(* CODESYS project full_demo.190528.1.project

Project tree, tasks and I/O mapping:
  MIC7001 : Changsha Xiangji-ARM Cortex A9(xilinx zynq7000)-linux, Changsha Xiangji Hiden Technology Co.Ltd, version 3.5.10.40
    application Application
      libraries: Standard, * (System); CAA File, * (CAA Technical Workgroup); CAA Types Extern, * (CAA Technical Workgroup); CAA Callback Extern, * (CAA Technical Workgroup); SysMem, * (System); Util, 3.5.11.0 (System); SysFile, 3.5.9.0 (System); SysTypes Interfaces, * (System); CAN API, 1.0.0.3 (3S - Smart Software Solutions GmbH); SysTime, * (System); CAA DTUtil Extern, 3.5.12.0 (CAA Technical Workgroup); CAA SerialCom, 3.5.12.0 (CAA Technical Workgroup); cyber gpio, 3.5.10.40 (cyber); AC_DataLog, 3.5.13.0 (3S - Smart Software Solutions GmbH)
      task MainTask (cyclic, interval 20 ms, priority 15) calls prg_input, prg_engine, prg_pump, prg_output, prg_data
      task can_0 (cyclic, interval 8 ms, priority 10) calls prg_can0
      task VISU_TASK (cyclic, interval 100 ms, priority 31) calls VisuElems.Visu_Prg, prg_set_inmode, prg_heartbeat
      task EtherCAT_Task (cyclic, interval t#4ms, priority 1) calls nothing
      program prg_pump [ST]
      program prg_output [ST]
      program prg_input [ST]
      j1939/
        function temp_absZero_to_1735oC [ST]
        function block PGN_F004_RPM [ST]
        function pros100 [ST]
        function block PGN_FEEE_TEMP [ST]
        function temp_neg40_to_210oC [ST]
        function PACK [ST]
      program prg_can0 [CFC]: act_set_rpm, act_send_to_MID
      function_blocks/
        function block MsgProcessor_j1939_f004 [ST]: ProcessMessage
        function block fb_pp_avg [ST]
        function block MsgProcessor_j1939_f003 [ST]: ProcessMessage
        function block MsgProcessor_MID [ST]: ProcessMessage
        function block MsgProcessor_j1939_fef2 [ST]: ProcessMessage
        function block MsgProcessor_j1939_feef [ST]: ProcessMessage
        function block MsgProcessor_j1939_feee [ST]: ProcessMessage
      program prg_set_inmode [ST]
      ENUM/
        data type ENGINE_STATE
        data type STATE1939
        data type WORK_MODE
      global variables GVL
      parameters/
        function block FB_PARA_DINT [ST]: clear_all, rd_all, chk_chg, wr_all
        data type DUT_PARA_DINT
        data type DUT_PARA_REAL
        function block FB_PARA_REAL [ST]: rd_all, chk_chg, clear_all, wr_all
      functions/
        function fn_write_in_mode_file [ST]
        function fn_write_real_data [ST]
        function fn_read_in_mode_file [ST]
        function fn_get_Q_221ma [ST]
        function fn_get_Q_408ma [ST]
        function fn_get_Q_631ma [ST]
        function fn_get_Q_521ma [ST]
        function fn_write_dint_data [ST]
        function fn_get_mins [ST]
      program prg_data [ST]
      visualisation Visualization
      program prg_engine [ST]: get_x_rpm_set
      GPRS/
        function block File_Read [ST]
        function Iccid_Get [ST]
        program prg_heartbeat [ST]
        function block fb_get_iccid [ST]
        function block fb_m26 [ST]
        function block fb_get_lac [ST]
        function fn_cyber_layer1 [ST]
        function fn_cyber_layer2 [ST]
        function fn_cyber_heartBeat [ST]
        function fn_sn_str_to_byte [ST]
      gprs_lib/
        function block Com_Read [ST]
        function block reset_gprs [ST]
        function block Udp_Config [ST]
        function block Udp_Init [ST]
        function block UDP_Read [ST]
        function block Udp_Write [ST]
    EtherCAT_Master_SoftMotion : EtherCAT Master SoftMotion, 3S - Smart Software Solutions GmbH, version 3.5.13.30
        settings: NetworkName = 'eth0'; NetworkName = "eth0"; SelectNetworkByName = True
      MIR3502 : MIR3502, Cyber-MI, order no. MIR3502, version Revision=16#00000000
          settings: DC sync0 cycletime = 4000; DC sync1 cycletime = 4000
          unmapped channels: PWM00-C24, PWM01-C35, DO00-C01, DO01-C02, DO02-C03, DO03-C04, DO04-C05, DO05-C06, DO06-C07, DO07-C08, DO08-C09, DO09-C10, DO10-C11, DO11-C12, DO12-C35, DO13-C34, DO14-C33, DO15-C32, DO16-C31, DO17-C30, DO18-C29, DO19-C28, DO20-C27, DO21-C26, DO22-C25, DO23-C24, AI00-C20, AI01-C19, AI02-C18, AI03-C17, AI04-C16, AI05-C15, AI06-C01, AI07-C02, AI08-C03, AI09-C04, AI10-C05, AI11-C06, AI12-C07, AI13-C08,
            AI14-C09, AI15-C10, AI16-C11, AI17-C12, AI18-C35, AI19-C34, AI20-C33, AI21-C32, AI22-C31, AI23-C30, AI24-C29, AI25-C28, AI26-C27, AI27-C26, AI28-C25, AI29-C24, AI30-iPWM0, AI31-iPWM1, DI00-C20, DI01-C19, DI02-C18, DI03-C17, DI04-C16, DI05-C15, DI06-C01, DI07-C02, DI08-C03, DI09-C04, DI10-C05, DI11-C06, DI12-C07, DI13-C08, DI14-C09, DI15-C10, DI16-C11, DI17-C12, DI18-C35, DI19-C34, DI20-C33, DI21-C32,
            DI22-C31, DI23-C30, DI24-C29, DI25-C28, DI26-C27, DI27-C26, DI28-C25, DI29-C24, DI30, DI31
    SoftMotion General Axis Pool
    IoDrvMIC7001 : IoDrvMIC7001, MyCompany, version 19.1.1
        input  Application.GVL.AI_pilot : DWORD  // Ai00@C16
        input  Application.GVL.AI_pump1 : DWORD  // Ai01@C28
        input  Application.GVL.AI_pump2 : DWORD  // Ai02@C17
        input  Application.GVL.AI_grade : DWORD  // Ai03@C29
        input  Application.GVL.AI_oil_water : DWORD  // Ai05@C19
        input  Application.GVL.AI_temp_oil : DWORD  // Ai28-Do10@C10
        input  Application.GVL.AI_fuel_level : DWORD  // Ai46-Ao00@C22
        input  Application.gvl.AI_vcc : DWORD  // Ai50_VCC
        input  Application.gvl.AI_curr_prop : DWORD  // Ai53_Pwm-i0
        input  Application.GVL.DI_air_filter : BOOL  // Di06-Ai06@C31
        input  Application.GVL.DI_idle_button : BOOL  // Di07-Ai07@C20
        input  Application.GVL.DI_start : BOOL  // Di08-Ai08@C18
        input  Application.GVL.DI_high_power : BOOL  // Di24-Ai24@C05
        input  Application.GVL.DI_pilot : BOOL  // Di25-Ai25@C06
        input  Application.GVL.DI_work : BOOL  // Di26-Ai26@C08
        input  Application.GVL.DI_move : BOOL  // Di27-Ai27@C09
        output Application.GVL.DO_stop : BOOL  // Do00-Ai18@C25
        output Application.GVL.DO_pilot : BOOL  // Do01-Ai19@C24
        output Application.GVL.DO_high_power : BOOL  // Do02-Ai20@C13
        output Application.GVL.DO_high_speed : BOOL  // Do03-Ai21@C01
        output Application.GVL.DO_start : BOOL  // Do04-Ai22@C03
        output Application.GVL.DO_dump_load : BOOL  // Do05-Ai23@C04
        output Application.GVL.PWM_prop : DWORD  // PWM28-Pwmi00@C33
        output Application.gvl.do_led_run : BOOL  // LED_run
        output Application.gvl.DO_led_err : BOOL  // LED_err
        output Application.gvl.DO_led_usr : BOOL  // LED_usr
        unmapped channels: Ai04@C30, Ai06@C31, Ai07@C20, Ai08@C18, Ai09@D18, Ai10@D20, Ai11@D31, Ai12@D19, Ai13@D30, Ai14@D29, Ai15@D17, Ai16@D28, Ai17@D16, Ai18-Do00@C25, Ai19-Do01@C24, Ai20-Do02@C13, Ai21-Do03@C01, Ai22-Do04@C03, Ai23-Do05@C04, Ai24-Do06@C05, Ai25-Do07@C06, Ai26-Do08@C08, Ai27-Do09@C09, Ai29-Do11@C11, Ai30-Do12@D34, Ai31-Do13@D35, Ai32-Do14@D23, Ai33-Do15@D12, Ai34-Do16@D10, Ai35-Do17@D09, Ai36-Do18@D08, Ai37-Do19@D07, Ai38-Do20@D05, Ai39-Do21@D04, Ai40-Do22@D03, Ai41-Do23@D02, Ai42-Do24@C23, Ai43-Do25@C35, Ai44-Do26@D24, Ai45-Do27@D13,
          Ai47-Ao01@D14, Ai48_Pi02, Ai49_Out5V, Ai51_VCC_L, Ai52_VCC_R, Ai54_Pwm-i1, Ai55_Pwm-i2, Ai56_Pwm-i3, Ai57_CPU-T, Ai58_G-x, Ai59_G-y, Ai60_G-z, Ai61-reserved, Ai62-IO-cntr, Ai63-CDS-cntr, Di00-Ai00@C16, Di01-Ai01@C28, Di02-Ai02@C17, Di03-Ai03@C29, Di04-Ai04@C30, Di05-Ai05@C19, Di09-Ai09@D18, Di10-Ai10@D20, Di11-Ai11@D31, Di12-Ai12@D19, Di13-Ai13@D30, Di14-Ai14@D29, Di15-Ai15@D17, Di16-Ai16@D28, Di17-Ai17@D16, Di18-Ai18@C25, Di19-Ai19@C24, Di20-Ai20@C13, Di21-Ai21@C01, Di22-Ai22@C03, Di23-Ai23@C04, Di28-Ai28@C10, Di29-Ai29@C11, Di30-Ai30@D34, Di31-Ai31@D35,
          Di32-Ai32@D23, Di33-Ai33@D12, Di34-Ai34@D10, Di35-Ai35@D09, Di36-Ai36@D08, Di37-Ai37@D07, Di38-Ai38@D05, Di39-Ai39@D04, Di40-Ai40@D03, Di41-Ai41@D02, Di42-Ai42@C23, Di43-Ai43@C35, Di44-Ai44@D24, Di45-Ai45@D13, Di46-Ai46@C22, Di47-Ai47@D14, Di48-Pi00@C15, Di49-Pi01@C14, Di50-Pi02@D22, Di51-Pi03@D21, Di52-reserved, Di53-reserved, Di54-reserved, Di55-reserved, Di56-reserved, Di57-reserved, Di58-reserved, Di59-reserved, Di60-reserved, Di61-reserved, Di62-reserved, Di63-reserved, Pi00-Di48@C15, Pi01-Di49@C14, Pi02-Di50@D22, Pi03-Di51@D21, Do06-Ai24@C05, Do07-Ai25@C06, Do08-Ai26@C08, Do09-Ai27@C09,
          Do10-Ai28@C10, Do11-Ai29@C11, Do12-Ai30@D34, Do13-Ai31@D35, Do14-Ai32@D23, Do15-Ai33@D12, Do16-Ai34@D10, Do17-Ai35@D09, Do18-Ai36@D08, Do19-Ai37@D07, Do20-Ai38@D05, Do21-Ai39@D04, Do22-Ai40@D03, Do23-Ai41@D02, Do24-Ai42@C23, Do25-Ai43@C35, Do26-Ai44@D24, Do27-Ai45@D13, Do28-Pwmi00@C33, Do29-Pwmi01@C34, Do30-Pwmi02@D25, Do31-Pwmi03@D26, PWM00@C25, PWM01@C24, PWM02@C13, PWM03@C01, PWM04@C03, PWM05@C04, PWM06@C05, PWM07@C06, PWM08@C08, PWM09@C09, PWM10@C10, PWM11@C11, PWM12@D34, PWM13@D35, PWM14@D23, PWM15@D12, PWM16@D10, PWM17@D09,
          PWM18@D08, PWM19@D07, PWM20@D05, PWM21@D04, PWM22@D03, PWM23@D02, PWM24@C23, PWM25@C35, PWM26@D24, PWM27@D13, PWM29-Pwmi01@C34, PWM30-Pwmi02@D25, PWM31-Pwmi03@D26, PWM_I_0@C33, PWM_I_1@C34, PWM_I_2@D25, PWM_I_3@D26, Ao00-Ai46@C22, Ao01-Ai47@D14, ctrl_ai_raw, ctrl_adjust, ctrl_adj0, ctrl_adj1, ctrl_adj2, ctrl_adj3, ctrl_adj4
  text list GlobalTextList
*)

// MIC7001/Application/ENUM/ENGINE_STATE
TYPE ENGINE_STATE : 
(
	PWR_OFF := 0, 	(* 断电状态 *)
	PWR_ON,		(* 上电状态 *)
	START_FAIL,	(* 启动失败 *)
	START_IDLE,	(* 启动后低速运行 *)
	START_RUN,  (* 启动后短时升速*)
	RUNNING,	(* 正常运行*)
	ADJUSTING,	(* 档位校准*)
	RUN_IDLE,	(* 自动怠速*)
	STOPPING	(* 正在熄火*)
);
END_TYPE

// MIC7001/Application/ENUM/STATE1939
{attribute 'qualified_only'}
{attribute 'strict'}
TYPE STATE1939 :
(
	INIT := 0, 	(* first State. Connections are set up *)
	SEND,		(* Send messages *)
	READ,		(* Receive messages *)
	ERROR		(* Prepare to reset connections *)
);
END_TYPE

// MIC7001/Application/parameters/DUT_PARA_DINT
TYPE DUT_PARA_DINT :
STRUCT
	num:UINT := 64;  //可根据需要设置总数量，最后一个为校验和，不可用
	para:ARRAY[1..64] OF DINT;  //三行中的总数量需要严格一致
	old_val:ARRAY[1..64] OF DINT; //三行中的总数量需要严格一致
	filename :STRING := 'mic_dint.txt';  
END_STRUCT
END_TYPE

// MIC7001/Application/ENUM/WORK_MODE
TYPE WORK_MODE : 
(
	STANDARD := 0, 	(* 标准模式 *)
	HEAVY,		(* 重载模式 *)
	LIGHT,		(* 轻载模式 *)
	INTELLIGENT (*智能模式*)
);
END_TYPE

// MIC7001/Application/parameters/DUT_PARA_REAL
TYPE DUT_PARA_REAL :
STRUCT
	num:UINT := 256; //可根据需要设置总数量，最后一个为校验和，不可用
	para:ARRAY[1..256] OF REAL;  //三行中的总数量需要严格一致
	old_val:ARRAY[1..256] OF REAL; //三行中的总数量需要严格一致
	filename :STRING := 'mic_real.txt';  
END_STRUCT
END_TYPE

// MIC7001/Application/GVL
VAR_GLOBAL
	g_pump_work:BOOL := TRUE;  //液压泵软开关
	g_engine_work:BOOL := TRUE;  //发动机软开关
	
	//小时计相关
	g_running_mins:DINT := 0; //控制器运行的分钟数
	g_machine_start_mins:DINT := 0; //主机出厂时对应的控制器分钟数，需要放在掉电保持的参数区
	g_machine_mins:DINT := 0; //主机运行的分钟数, = g_running_mins - g_machine_start_mins
	g_engine_mins:DINT := 0; //发动机运行的分钟数
	
	g_machine_mins_1_start:DINT := 0; //阶段小时计1开始时间
	g_machine_mins_2_start:DINT := 0; //阶段小时计2开始时间
	
	g_machine_mins_1:DINT := 0;
	g_machine_mins_2:DINT := 0;
	
	// PORT CAN1 GLOBAL HANDLE
	g_hCan1939: CAA.HANDLE ;
	g_hRecv_FEEE: CAA.HANDLE := 0;
	g_hRecv_FEEF: CAA.HANDLE := 0;
	g_hRecv_F003: CAA.HANDLE := 0;
	g_hRecv_F004: CAA.HANDLE := 0;
	g_hRecv_18F: CAA.HANDLE := 0;
	
	//发动机相关实时数据
	g_P_KW_max:DINT := 30;  //当前发动机储备功率
	g_rpm_set: DINT := 1000;  //当前设定转速
	g_rpm_real: DINT := 0; //当前实时转速
	g_fuel_rate_1939:REAL := 0; //从发动机读到的瞬时油耗，单位：ml/s
	g_temp_coolant_1939:REAL := 0; //从发动机读到的水温， 单位：摄氏度
	g_oil_press_1939:REAL := 0; //从发动机读到的机油压力， 单位： kPa
	g_coolant_level_1939:REAL := 0; //从发动机读到的冷却液液位， 单位： 百分比
	g_load_percent_1939:REAL := 0; //从发动机读到的发动机负载率， 单位： 百分比
	g_demand_torque_1939:REAL := 0; //从发动机读到的需求扭矩， 单位： 百分比
	g_real_torque_1939:REAL := 0; //从发动机读到的实际扭矩， 单位：百分比
	
	g_x_duty_min :REAL := 0.25;
	g_x_duty_max :REAL := 0.75;
	
	//统计数据
	g_fuel_depleted: DINT;  //出厂累计油耗，单位：升
	g_fuel_depleted_1: DINT; //阶段一累计油耗，单位：升 
	g_fuel_depleted_2: DINT; //阶段二累计油耗，单位：升
	
	
	g_Eng_Coolaant_Temp:INT;(*spn 110*)
	g_Eng_Fuel_Temp:INT;(*spn 174*)
	g_Eng_Oil_Temp:INT;(*spn 175*)
	g_Turbo_Oil_Temp:INT;(*spn 176*)
	g_Eng_InterCooler_Temp:INT;(*spn 52*)
	g_Eng_InterCooler_Thermostat_Opening:BYTE;(*spn 1134*)
	
	g_mode: WORK_MODE := STANDARD; //working mode  
						//0:Standard  	标准模式  
						//1:Heavy   	重载模式
						//2:Light  		轻载模式
						//3:Break		破碎模式
						
	g_res_prop:REAL := 20; //电磁比例阀电阻，动态调整

	//熟数据
	g_ai_press_pump1:REAL;
	g_ai_press_pump1_trace:REAL;
	g_ai_press_pump2:REAL;
	g_ai_press_pump2_trace :REAL;
	g_ai_pilot:REAL;
	g_ai_pilot_trace: REAL;
	g_ai_curr_prop:UINT;
	g_ai_curr_prop_trace:REAL;
	g_ai_oil_water:BOOL;
	g_ai_vcc:DWORD;
	g_ai_fuel_level:REAL;

	g_di_start:BOOL := FALSE; //上电信号
	g_di_move:BOOL := FALSE; //工作装置压力开关
	g_di_work:BOOL := FALSE; //行走压力开关
	g_di_pilot:BOOL := FALSE;  //先导手柄开关输入
	
	g_do_start:BOOL := TRUE;  //启动继电器		
	g_do_ecu:BOOL := TRUE;    //为true为发动机ECU供电
	g_do_pilot:BOOL := FALSE;
	
	g_pwm_prop:DINT := 0; 
	
	g_rpm_trace:REAL := 0;  //示波器变量，转换到0~10之间
	//间接计算数据
	g_psp: REAL := 0;   //电磁比例阀二次压力  MPa
	g_backup_power:REAL := 0;   //发动机储备功率  KW
	g_backup_power_trace:REAL; //示波器变量，转换到0~10之间
	g_duty_power:REAL := 0; //发动机功率利用率
	g_backup_torque:REAL := 0;  //发动机储备扭矩  N*M
	g_backup_torque_trace:REAL;//示波器变量，转换到0~10之间
	g_duty_torque:REAL := 0;  //发动机扭矩利用率
	g_flow1 :REAL := 0;   //前泵流量 L/min
	g_flow1_trace:REAL;//示波器变量，转换到0~10之间
	g_flow2 :REAL := 0;   //后泵流量 L/min
	g_flow2_trace:REAL;//示波器变量，转换到0~10之间
	g_power_pump1 :REAL := 0;   //前泵功率  KW
	g_power_pump1_trace:REAL;//示波器变量，转换到0~10之间
	g_power_pump2 :REAL := 0;   //后泵功率  KW
	g_power_pump2_trace:REAL;//示波器变量，转换到0~10之间
	g_torque_pump1 :REAL := 0;  //前泵输出扭矩  N*M
	g_torque_pump2 :REAL := 0;  //后泵输出扭矩  N*M
	
// I/O port mapping var
	AI_pump1:DWORD; //前泵压力
	AI_pump2:DWORD; //后泵压力
	AI_pilot:DWORD; //先导压力
	AI_curr_prop:DWORD; //电磁比例阀电流
	AI_oil_water:DWORD; //油水分离器
	AI_vcc:DWORD; //电源电压 mV
	AI_grade:DWORD; //油门旋钮
	AI_temp_oil:DWORD; //液压油温
	AI_fuel_level:DWORD; //液位传感器
		
	
	DI_start: BOOL; //启动信号
	DI_pilot:BOOL; //先导手柄闭合
	DI_move:BOOL; //行走压力开关
	DI_work:BOOL; //作业压力开关
	DI_air_filter:BOOL;  //空滤堵塞
	DI_idle_button:BOOL;  //机械怠速按钮
	DI_high_power:BOOL; //增力信号输入
	
	
	DO_start: BOOL := FALSE; //驱动启动电机
	DO_stop: BOOL := TRUE;  //驱动熄火继电器
	DO_pilot :BOOL := TRUE;  //驱动先导阀
	DO_high_power:BOOL := FALSE; //增力输出
	DO_high_speed:BOOL := FALSE; //高速输出
	DO_dump_load:BOOL := FALSE; //卸载输出
	
					
	PWM_prop:DWORD; //油泵电磁比例阀	
	
	RPM_engine:UINT; //柴油机转速  J1939

	DO_led_run:BOOL;
	DO_led_err:BOOL;
	DO_led_usr:BOOL;
	
// 档位校准	
	adj_gear: BOOL := FALSE;  //校准档位旋钮
	gear_grade: UINT := 1;   //档位旋钮对应的档位
	running_grade:UINT := 1;  //当前实际运行的档位
	
	g_grade: DINT;	  //发动机档位
	//各档位对应的转速
	grade_rpm : ARRAY [1..10] OF DINT := [1200, 1350, 1450, 1550, 1650, 1750, 1850, 1950, 2050, 2100];
	
	//各档位对应的旋钮采样值（mV）
	grade_mv: ARRAY[1..10] OF DINT := [1534, 1705, 1876, 2056, 2242, 2439, 2625, 2810, 2988, 3168];

//显示屏发送来的命令
	cmd_auto_idle : BOOL := TRUE;
	cmd_high_speed: BOOL := FALSE;	
	cmd_more_power: BOOL := FALSE;
	cmd_clear_hours : BOOL := FALSE;
	cmd_clear_hours_1 :BOOL := FALSE;
	cmd_clear_hours_2 :BOOL := FALSE;
	
	//各模式的比例阀电流值
	pwm_of_mode_h : DINT := 580;  //H模式
	pwm_of_mode_s : DINT := 520;  //S模式
	pwm_of_mode_l : DINT := 490;  //L模式
	
	C_RPM_MIN: DINT := 800;
	C_RPM_IDLE: DINT := 1450;
	C_RPM_MAX : DINT := 2300;
	
	C_H_MAX_RPM: DINT := 2200;
	C_S_MAX_RPM: DINT := 2050;
	C_L_MAX_RPM: DINT := 1900;
	
	g_time_good: BOOL := FALSE;  //控制器本地时钟校准完成
END_VAR

VAR_GLOBAL CONSTANT
	inmode_file:STRING:='in_mode.txt';
	mins_file :STRING := '/userapp/r_mins.txt';
END_VAR

// MIC7001/Application/prg_input
PROGRAM prg_input
VAR

END_VAR


//先导油路安全开关输入
GVL.g_di_pilot := GVL.DI_pilot;

//电磁比例阀反馈电流计算
IF gvl.AI_curr_prop < 110 THEN
	gvl.g_ai_curr_prop := ANY_TO_UINT(gvl.AI_curr_prop)*200/110;
elsIF gvl.AI_curr_prop < 223 THEN
	gvl.g_ai_curr_prop := ANY_TO_UINT(gvl.AI_curr_prop-110)*50/56 + 200;
ELSE
	gvl.g_ai_curr_prop := ANY_TO_UINT(gvl.AI_curr_prop-223)*50/56 + 303;
END_IF
GVL.g_ai_curr_prop_trace := ANY_TO_REAL(GVL.g_ai_curr_prop)/1000.0;

//先导压力信号计算
IF GVL.AI_pilot < 4000 THEN
	GVL.g_ai_pilot := 0;
ELSE
	GVL.g_ai_pilot := ANY_TO_REAL(GVL.AI_pilot-4000)*6.0/(20000.0-4000.0);
END_IF
GVL.g_ai_pilot_trace := GVL.g_ai_pilot/10;

//前泵主压计算
IF GVL.AI_pump1 < 4000 THEN
	gvl.g_ai_press_pump1 := 0.0;
ELSE
	gvl.g_ai_press_pump1 := ANY_TO_REAL(gvl.AI_pump1-4000)*40.0/(20000.0-4000.0);
END_IF
GVL.g_ai_press_pump1_trace := GVL.g_ai_press_pump1/100;

//后泵主压计算
IF GVL.AI_pump2 < 4000 THEN
	gvl.g_ai_press_pump2 := 0.0;
ELSE
	gvl.g_ai_press_pump2 := ANY_TO_REAL(gvl.AI_pump2-4000)*40.0/(20000.0-4000.0);
END_IF
GVL.g_ai_press_pump2_trace := GVL.g_ai_press_pump2/100;

//电源电压计算
gvl.g_ai_vcc := gvl.AI_vcc;

//输入开关量信号
gvl.g_di_start := gvl.DI_start;  //启动输入信号
gvl.g_di_move := gvl.DI_move;
gvl.g_di_work := gvl.DI_work;

END_PROGRAM

// MIC7001/Application/prg_engine
PROGRAM prg_engine

VAR
	stat : ENGINE_STATE := PWR_OFF;
	timer_start:ton;
	flag_idle: BOOL;
	flag_stop: BOOL;
	rpm_max :DINT;
	rpm_max_heavy : DINT := 2100;
	rpm_max_standard : DINT := 2000;
	rpm_max_light : DINT := 1850;
	rpm_max_x : DINT := 2100;
	rpm_min_x : DINT := 1400;
	rpm_min :DINT := 1250;
	rpm_x: DINT := 1500;
	
	stat_gear:DINT := 1;
	old_grade: DINT;
	
	tmr_idle:ton;
END_VAR


CASE stat OF
	PWR_OFF: //停机状态
		IF gvl.g_di_start AND g_engine_work THEN
			stat := PWR_ON; 
			gvl.g_do_start := TRUE;
			timer_start(in := FALSE);
		END_IF
	
	PWR_ON: //上电状态
		IF g_rpm_real > C_RPM_MIN THEN   //start succeed
			stat := START_IDLE; //启动怠速
			gvl.g_do_start := TRUE;  //启动控制继电器
			gvl.g_do_ecu := TRUE;   //熄火继电器，常开触点为发动机ECU供电
			old_grade := gvl.gear_grade;
		END_IF
	
	START_FAIL:  //启动失败
		timer_start(in := TRUE,pt := T#5S);  //stop for 5 seconds to protect battery
		IF timer_start.Q THEN
			stat := PWR_ON;
		END_IF
		
	START_IDLE:  //启动怠速, 刚启动，不管油门旋钮的位置在哪里， 先运行在1档
		gvl.running_grade := 1;
		IF old_grade <> gvl.gear_grade THEN  //操作手调整档位
			old_grade := gvl.gear_grade;
			stat := RUNNING; //正常工作模式
		END_IF
		
		IF gvl.g_di_move OR gvl.g_di_work THEN
			stat := START_RUN;
		END_IF
		
	START_RUN:  //启动时短时升速运行,便于临时动作
		gvl.running_grade := 3;
		IF NOT gvl.g_di_move AND  NOT gvl.g_di_work THEN
			stat := START_IDLE;
		END_IF
		
	RUNNING:  //正常工作
		gvl.running_grade := gvl.gear_grade;
		IF flag_idle THEN
			stat := RUN_IDLE;
		END_IF	
		
		IF flag_stop THEN
			stat := STOPPING;
		END_IF		
		
		IF NOT g_engine_work THEN  //软件停机
			stat := STOPPING;
		END_IF
	RUN_IDLE:  //idle, running at 3 grade
		IF gvl.gear_grade > 3 THEN
			gvl.running_grade := 3;
		ELSE
			gvl.running_grade := gvl.gear_grade;
		END_IF
		
		IF NOT flag_idle THEN
			stat := RUNNING; //to running status
		END_IF
		
		IF NOT gvl.g_di_start THEN
			stat := STOPPING;
		END_IF
		
		IF NOT g_engine_work THEN  //软件停机
			stat := STOPPING;
		END_IF		
	STOPPING:  //stopping
		//gvl.g_do_ecu := FALSE;
		IF g_rpm_real < C_RPM_MIN THEN
			gvl.g_do_ecu := FALSE;
			stat := PWR_OFF;
		END_IF
END_CASE

//根据档位取得对应转速
gvl.g_rpm_set := gvl.grade_rpm[gvl.running_grade];

//根据设定的模式取得最大和最小转速
CASE g_mode OF
	STANDARD: 
		rpm_max := rpm_max_standard;
	HEAVY: 
		rpm_max :=rpm_max_heavy;
	LIGHT:
		rpm_max := rpm_max_light;
	INTELLIGENT:
		rpm_min_x := gvl.g_rpm_set - 300; //在300 转的范围内自动调整
		rpm_max := gvl.g_rpm_set;
		
		rpm_x := get_x_rpm_set(rpm_x);	
		gVL.g_rpm_set := rpm_x;	
		
		IF GVL.g_rpm_set < rpm_min_x THEN
			GVL.g_rpm_set := rpm_min_x;
		END_IF
END_CASE

IF gvl.g_rpm_set > rpm_max THEN
	gvl.g_rpm_set := rpm_max;
ELSIF GVL.g_rpm_set < rpm_min THEN
	GVL.g_rpm_set := rpm_min;
END_IF

//自动怠速条件判断
IF gvl.cmd_auto_idle=FALSE OR  gvl.g_di_move OR gvl.g_di_work THEN
	flag_idle := FALSE;
	tmr_idle(in := FALSE);
ELSE
	tmr_idle(in := TRUE, pt := T#3S);
	IF tmr_idle.Q THEN
		tmr_idle(in := FALSE, pt := T#3S);
		flag_idle := TRUE;
	END_IF
END_IF

//档位旋钮校准
IF NOT gvl.adj_gear THEN
	stat_gear := 1;
END_IF

METHOD get_x_rpm_set : DINT
VAR_INPUT
	rpm_old:DINT;
END_VAR

VAR
	old_duty_power :REAL := 0.25;
	rpm :DINT;
END_VAR
rpm := rpm_old;

IF g_duty_power > gvl.g_x_duty_max THEN
	rpm := rpm_old + 100;
ELSIF g_duty_power < GVL.g_x_duty_min THEN
	rpm := rpm_old - 1;
END_IF

rpm_old := rpm;

IF rpm > rpm_max_x THEN
	rpm := rpm_max_x;
ELSIF rpm < rpm_min_x THEN
	rpm := rpm_min_x;
END_IF

get_x_rpm_set := rpm;
END_METHOD

END_PROGRAM

// MIC7001/Application/prg_pump
PROGRAM prg_pump  //油泵比例阀电流调节
VAR
	wk_mode: WORK_MODE;
	current_of_pump: DINT;
	lead_press: REAL;
	vcc_pwm: UDINT;
	curr_pwm_max: REAL;
	pwm_val : DWORD := 0;
	ai_val: DWORD;
	curr_prog_ma: UINT;
	old_current_of_pump: DINT := 0;
	cntr_current_not_change: UDINT := 0;
	fb_pp:fb_pp_avg;
	old_pp:REAL := 3.0;  //上一次先导压力值
	pwm_of_mode_x : DINT := 520;  //X模式
	ton_idle:TON;
END_VAR

VAR CONSTANT
	PP_MIN:REAL := 3.5;  //最小先导压力
	PP_MAX:REAL := 4.0;  //最大先导压力
END_VAR


//根据设定的模式取得目标电流(mA)	
CASE g_mode OF
	STANDARD: 
		current_of_pump := gvl.pwm_of_mode_s;
	HEAVY: 
		current_of_pump := gvl.pwm_of_mode_h;
	LIGHT:
		current_of_pump := gvl.pwm_of_mode_l;
	INTELLIGENT:
		current_of_pump := pwm_of_mode_x;
END_CASE

IF GVL.g_di_move OR GVL.g_di_work THEN
	ton_idle(IN := FALSE, PT := T#1S);
END_IF
ton_idle(IN := TRUE, PT := T#1S);
IF ton_idle.Q THEN
	current_of_pump := 200;
END_IF


GVL.g_do_pilot := NOT GVL.g_di_pilot;

//计算100%占空比时的比例阀电流  单位： mA
curr_pwm_max := ANY_TO_REAL(gvl.g_ai_vcc)/g_res_prop; // 电源电压(mV)除以比例阀电阻(欧姆）
IF curr_pwm_max < 700 THEN
	curr_pwm_max := 700;
END_IF

IF GVL.running_grade < 4 THEN
	current_of_pump := 200;
END_IF

//计算比例阀PWM占空比
gvl.g_pwm_prop := 4096*ANY_TO_DINT(current_of_pump)/ANY_TO_DINT(curr_pwm_max);

//判断设定电流是否发生变化，用于后面的电阻校准
IF ABS(old_current_of_pump - current_of_pump) < 5 THEN
	cntr_current_not_change := cntr_current_not_change +1;
	IF cntr_current_not_change > 10000 THEN
		cntr_current_not_change := 10000;
	END_IF
ELSE
	cntr_current_not_change := 0;
END_IF
old_current_of_pump := current_of_pump;

//根据反馈电流与设定电流的差值，动态调整比例阀电阻
curr_prog_ma := gvl.g_ai_curr_prop;  
IF cntr_current_not_change > 50 AND current_of_pump>0   THEN //500 ms
	IF curr_prog_ma < current_of_pump - 5 THEN // 实际电流小于设定电流， 原电阻设定值偏小，需要增加
		g_res_prop := g_res_prop + 0.1;
		IF g_res_prop > 80 THEN
			g_res_prop := 80;
		END_IF
	ELSIF curr_prog_ma > current_of_pump + 5 THEN
		g_res_prop := g_res_prop - 0.1;
		IF g_res_prop < 5 THEN
			g_res_prop := 5;
		END_IF
	END_IF
END_IF

END_PROGRAM

// MIC7001/Application/function_blocks/fb_pp_avg
FUNCTION_BLOCK fb_pp_avg
VAR_INPUT
	pp:REAL; //当前先导压力
	flag_move:BOOL; //行走压力开关
	flag_work:BOOL; //工作装置压力开关
END_VAR
VAR_OUTPUT
	pp_avg_out:real := 3.0;  //计算结果
END_VAR
VAR
	pp_avg:REAL := 3.0;  //初始先导压力
END_VAR

IF NOT (flag_move OR flag_work) THEN   // 没有动作，不计算
	RETURN;
END_IF

pp_avg_out := pp_avg*0.95 + pp*0.05;

pp_avg := pp_avg_out;

END_FUNCTION_BLOCK

// MIC7001/Application/prg_output
PROGRAM prg_output
VAR
	ton_run:TON;
END_VAR

ton_run(IN := NOT ton_run.Q, PT := T#500MS);
IF ton_run.Q THEN
	gvl.DO_led_run := NOT gvl.DO_led_run;
END_IF

IF gvl.g_pump_work THEN  //液压泵软开关
	gvl.PWM_prop := ANY_TO_DWORD(gvl.g_pwm_prop);
	gvl.DO_pilot := gvl.g_do_pilot;
ELSE
	gvl.PWM_prop := 0;
	gvl.DO_pilot := FALSE;
END_IF

IF gvl.g_engine_work THEN //柴油机软开关
	gvl.DO_start := NOT gvl.g_do_start;  // 启动控制继电器，使用反逻辑控制
	gvl.DO_stop := NOT gvl.g_do_ecu;
ELSE
	gvl.DO_start := TRUE;   //禁止启动
	GVL.DO_stop := TRUE;   //ECU失电
	gvl.g_rpm_set := 0;
END_IF

END_PROGRAM

// MIC7001/Application/prg_data
PROGRAM prg_data
VAR
	data_save:BOOL := FALSE;
	
	save_data:ARRAY[0 .. 31] OF REAL;
	hFile: RTS_IEC_HANDLE := RTS_INVALID_HANDLE;
	data_len:UINT := 12;
	i:UINT;
	
	dateandtime : DTU.GetDateAndTime;
	dtDT :DATE_AND_TIME;
	
	data_stat:UINT := 0;
	
	curr_time : DWORD;
	pr:RTS_IEC_RESULT;
	
	ton_mins:ton;  //用于小时计的1分钟定时器
	data_save_cntr: INT;
END_VAR
VAR_INPUT
	para_dint:DUT_PARA_DINT;
	retain_dint:FB_PARA_DINT;
END_VAR

//整数参数掉电存储
retain_dint(enable := TRUE, pPara := ADR(para_dint));
CASE data_stat OF
0:
	IF retain_dint.zero THEN
		FOR i:= 1 TO 10 DO
			para_dint.para[i] := gvl.grade_rpm[i];
			para_dint.para[10+i] := gvl.grade_mv[i];
		END_FOR
		
		para_dint.para[21] := gvl.pwm_of_mode_h;
		para_dint.para[22] := gvl.pwm_of_mode_s;
		para_dint.para[23] := gvl.pwm_of_mode_l;
		
		para_dint.para[24] := gvl.C_RPM_MIN;
		para_dint.para[25] := gvl.C_RPM_IDLE;
		para_dint.para[26] := gvl.C_RPM_MAX;
		
		para_dint.para[27] := gvl.C_H_MAX_RPM;;
		para_dint.para[28] := gvl.C_S_MAX_RPM;
		para_dint.para[29] := gvl.C_L_MAX_RPM;
		
		para_dint.para[30] := gvl.g_fuel_depleted;
		para_dint.para[31] := gvl.g_fuel_depleted_1;
		para_dint.para[32] := gvl.g_fuel_depleted_2;
		para_dint.para[33] := 0;
		
		para_dint.para[34] :=  gvl.g_running_mins;  //控制器总运行时间分钟数，不可清空
		para_dint.para[35] := gvl.g_machine_start_mins;  //主机运行的开始时间，可清零
		para_dint.para[36] := gvl.g_engine_mins;  //发动机运行的分钟数，不可清空
		para_dint.para[37] := gvl.g_machine_mins_1_start;  //主机运行阶段一开始时间，可清零
		para_dint.para[38] := gvl.g_machine_mins_2_start;  //主机运行阶段二开始时间，可清零
	
	ELSE
		FOR i:= 1 TO 10 DO
			gvl.grade_rpm[i] := para_dint.para[i];
			gvl.grade_mv[i] := para_dint.para[10+i];
		END_FOR
		gvl.pwm_of_mode_h := para_dint.para[21];
		gvl.pwm_of_mode_s := para_dint.para[22] ;
		gvl.pwm_of_mode_l := para_dint.para[23]  ;
		
		gvl.C_RPM_MIN := para_dint.para[24] ;
		gvl.C_RPM_IDLE := para_dint.para[25] ;
		gvl.C_RPM_MAX := para_dint.para[26] ;
		
		gvl.C_H_MAX_RPM := para_dint.para[27];
		gvl.C_S_MAX_RPM := para_dint.para[28];
		gvl.C_L_MAX_RPM := para_dint.para[29];
		
		gvl.g_fuel_depleted := para_dint.para[30];
		gvl.g_fuel_depleted_1 := para_dint.para[31];
		gvl.g_fuel_depleted_2 := para_dint.para[32];
//		gvl.C_X_MODE_RPM := para_dint.para[33];		

		gvl.g_running_mins := para_dint.para[34]   ;
		gvl.g_machine_start_mins := para_dint.para[35];
		
		gvl.g_engine_mins  := para_dint.para[36];
		gvl.g_machine_mins := gvl.g_running_mins - gvl.g_machine_start_mins;
		
		gvl.g_machine_mins_1_start  := para_dint.para[37];
		gvl.g_machine_mins_1 := gvl.g_running_mins - gvl.g_machine_mins_1_start;
		
		gvl.g_machine_mins_2_start  := para_dint.para[38];
		gvl.g_machine_mins_2 := gvl.g_running_mins - gvl.g_machine_mins_2_start;
		
		data_stat := 10;
	END_IF
10:
		FOR i:= 1 TO 10 DO
			para_dint.para[i] := gvl.grade_rpm[i];
			para_dint.para[10+i] := gvl.grade_mv[i];
		END_FOR
		
		para_dint.para[21] := gvl.pwm_of_mode_h;
		para_dint.para[22] := gvl.pwm_of_mode_s;
		para_dint.para[23] := gvl.pwm_of_mode_l;
		
		para_dint.para[24] := gvl.C_RPM_MIN;
		para_dint.para[25] := gvl.C_RPM_IDLE;
		para_dint.para[26] := gvl.C_RPM_MAX;
		
		para_dint.para[27] := gvl.C_H_MAX_RPM;;
		para_dint.para[28] := gvl.C_S_MAX_RPM;
		para_dint.para[29] := gvl.C_L_MAX_RPM;
		
		para_dint.para[30] := gvl.g_fuel_depleted;
		para_dint.para[31] := gvl.g_fuel_depleted_1;
		para_dint.para[32] := gvl.g_fuel_depleted_2;
		para_dint.para[33] := 0;
		
		para_dint.para[34] :=  gvl.g_running_mins;  //控制器总运行时间分钟数，不可清空
		para_dint.para[35] := gvl.g_machine_start_mins;  //主机运行的开始时间，可清零
		para_dint.para[36] := gvl.g_engine_mins;  //发动机运行的分钟数，不可清空
		para_dint.para[37] := gvl.g_machine_mins_1_start;  //主机运行阶段一开始时间，可清零
		para_dint.para[38] := gvl.g_machine_mins_2_start;  //主机运行阶段二开始时间，可清零
END_CASE

ton_mins(in := NOT ton_mins.Q, pt := T#60S);
IF ton_mins.Q THEN
	gvl.g_running_mins := gvl.g_running_mins + 1;
	para_dint.para[34] := gvl.g_running_mins;
	IF gvl.g_rpm_real > gvl.C_RPM_MIN THEN   //发动机在运行
		gvl.g_engine_mins := gvl.g_engine_mins + 1;
		para_dint.para[36] := gvl.g_engine_mins;
	END_IF
	
	gvl.g_machine_mins := gvl.g_running_mins - gvl.g_machine_start_mins;  //工作小时计
	gvl.g_machine_mins_1 := gvl.g_running_mins - gvl.g_machine_mins_1_start; //阶段小时计1
	gvl.g_machine_mins_2 := gvl.g_running_mins - gvl.g_machine_mins_2_start;  //阶段小时计2
END_IF

//保存实时数据
IF data_save = FALSE THEN   //停止写数据，关闭文件
	IF hFile <> RTS_INVALID_HANDLE THEN
		hFile := fn_write_dint_data(close := TRUE, num := data_len, hFile := hFile, pData := ADR(save_data));
		hFile := RTS_INVALID_HANDLE;
	END_IF
	data_save_cntr := 0;
ELSE
	data_save_cntr := data_save_cntr + 1;
	IF data_save_cntr > 30000 THEN  //tick = 20ms,   50 points/second,  30000 points /10 minutes
		data_save := FALSE;
	END_IF

	save_data[0] := ANY_TO_REAL(data_save_cntr); //记录序号
	save_data[1] := ANY_TO_REAL(gvl.g_ai_curr_prop);  //比例阀电流  mA
	save_data[2] := ANY_TO_REAL(gvl.g_ai_pilot); //先导压力  MPa
	save_data[3] := ANY_TO_REAL(gvl.g_ai_press_pump1); //前泵压力  MPa
	save_data[4] := ANY_TO_REAL(gvl.g_ai_press_pump2); //后泵压力 MPa
	save_data[5] := ANY_TO_REAL(gvl.g_flow1);  //前泵流量  L/min
	save_data[6] := ANY_TO_REAL(gvl.g_flow2);  //后泵流量  L/min
	save_data[7] := ANY_TO_REAL(gvl.g_pwm_prop); //比例阀占空比  %
	save_data[8] := ANY_TO_REAL(gvl.g_power_pump1);  //前泵功率 kw
	save_data[9] := ANY_TO_REAL(gvl.g_power_pump2);  //后泵功率 kw
	save_data[10] := ANY_TO_REAL(gvl.g_backup_power);   //功率储备  Kw
	save_data[11] := ANY_TO_REAL(gvl.g_torque_pump1); //前泵扭矩
	save_data[12] := ANY_TO_REAL(gvl.g_torque_pump2); //后泵扭矩
	save_data[13] := ANY_TO_REAL(gvl.g_backup_torque);  //扭矩储备  N*m
	save_data[14] := ANY_TO_REAL(gvl.g_load_percent_1939); //负载率  %
	save_data[15] := ANY_TO_REAL(gvl.g_demand_torque_1939); //需求扭矩  N*m
	save_data[16] := ANY_TO_REAL(gvl.g_real_torque_1939);  //实际扭矩  N*m	
	
	save_data[17] := ANY_TO_REAL(gvl.g_rpm_set);  //目标转速   RPM
	save_data[18] := ANY_TO_REAL(gvl.g_rpm_real);  //实际转速  RPM
	save_data[19] := ANY_TO_REAL(gvl.g_fuel_rate_1939);  //燃油率  ml/s
	save_data[20] := ANY_TO_REAL(gvl.g_temp_coolant_1939); //冷却液温度  ℃
	save_data[21] := ANY_TO_REAL(gvl.g_oil_press_1939);  //机油压力  KPa
	save_data[22] := ANY_TO_REAL(gvl.g_coolant_level_1939);  //冷却液位  %
	save_data[23] := ANY_TO_REAL(gvl.g_res_prop);  //比例阀电阻   Ω
	
	data_len := 24;  //根据上面数据调整  0~23 
	
	hFile := fn_write_real_data(close := FALSE, num := data_len, hFile := hFile, pData := ADR(save_data));
END_IF

END_PROGRAM

// MIC7001/Application/functions/fn_write_dint_data
FUNCTION fn_write_dint_data : RTS_IEC_HANDLE
VAR_INPUT
	pData: POINTER TO DINT := 0;
	num:UINT := 0;	
	close:BOOL:= FALSE;
	hFile: RTS_IEC_HANDLE := RTS_INVALID_HANDLE;
END_VAR

VAR
	udiDeleteError: RTS_IEC_RESULT;
	udiOpenError: RTS_IEC_RESULT;
	udiWriteError: RTS_IEC_RESULT;
	udiSizeError: RTS_IEC_RESULT;
	filesize: __XWORD;
	i :DWORD;
	iTemp: UDINT;
	udiPos: UDINT;
	str: STRING(256);
	str_size: __XWORD;
	udiByteWrite: LWORD;
	check_sum:REAL := 0;
	gRandomNum :LWORD := 1;   //系统随机数,每个周期乘以内部传感器的实时值；
	filename:STRING := 'running_data_dint.txt';
END_VAR

fn_write_dint_data := RTS_INVALID_HANDLE;

IF close THEN
	IF hFile <> RTS_INVALID_HANDLE THEN
		sysfileclose(hFile := hFile);
		hFile := RTS_INVALID_HANDLE;
	END_IF
	fn_write_dint_data := RTS_INVALID_HANDLE;
	RETURN;
END_IF

IF hFile = RTS_INVALID_HANDLE THEN
	hFile := sysfileopen(szFile := filename, am := sysfile.AM_APPEND_PLUS, pResult:= ADR(udiOpenError));
	IF hFile = RTS_INVALID_HANDLE	THEN  //打开文件失败
		RETURN;
	END_IF
END_IF

filesize := sysfilegetsize(filename, ADR(udiSizeError));
udiPos := SysFileSetPos(hFile:=hFile, ulOffset:=filesize);	

str:= '';
FOR i := 0 TO num-1 DO
	str := concat(str, DINT_TO_STRING(pData[i]));
	str := concat(str, ',');
END_FOR

str := concat(str, '$N');		
str_size := ANY_TO_DWORD(len(str));

udiByteWrite := sysfile.SysFileWrite(hFile := hFile,pbyBuffer := ADR(str),ulSize := str_size, pResult := ADR(udiWriteError));

fn_write_dint_data := hFile;   //保持打开状态，下次继续写入

END_FUNCTION

// MIC7001/Application/functions/fn_write_real_data
FUNCTION fn_write_real_data : RTS_IEC_HANDLE
VAR_INPUT
	pData: POINTER TO REAL := 0;
	num:UINT := 0;	
	close:BOOL:= FALSE;
	hFile: RTS_IEC_HANDLE := RTS_INVALID_HANDLE;
END_VAR

VAR
	udiDeleteError: RTS_IEC_RESULT;
	udiOpenError: RTS_IEC_RESULT;
	udiWriteError: RTS_IEC_RESULT;
	udiSizeError: RTS_IEC_RESULT;
	filesize: __XWORD;
	i :DWORD;
	iTemp: UDINT;
	udiPos: UDINT;
	str: STRING(256);
	str_size: __XWORD;
	udiByteWrite: LWORD;
	check_sum:REAL := 0;
	gRandomNum :LWORD := 1;   //系统随机数,每个周期乘以内部传感器的实时值；
	filename:STRING := 'running_data_real.csv';
END_VAR

fn_write_real_data := RTS_INVALID_HANDLE;

IF close THEN
	IF hFile <> RTS_INVALID_HANDLE THEN
		sysfileclose(hFile := hFile);
		hFile := RTS_INVALID_HANDLE;
	END_IF
	fn_write_real_data := RTS_INVALID_HANDLE;
	RETURN;
END_IF

IF hFile = RTS_INVALID_HANDLE THEN
	hFile := sysfileopen(szFile := filename, am := sysfile.AM_APPEND_PLUS, pResult:= ADR(udiOpenError));
	IF hFile = RTS_INVALID_HANDLE	THEN  //打开文件失败
		RETURN;
	END_IF
END_IF

filesize := sysfilegetsize(filename, ADR(udiSizeError));
udiPos := SysFileSetPos(hFile:=hFile, ulOffset:=filesize);	

str:= '';
FOR i := 0 TO num-1 DO
	str := concat(str, REAL_TO_STRING(pData[i]));
	str := concat(str, ',');
END_FOR

str := concat(str, '$N');		
str_size := ANY_TO_DWORD(len(str));

udiByteWrite := sysfile.SysFileWrite(hFile := hFile,pbyBuffer := ADR(str),ulSize := str_size, pResult := ADR(udiWriteError));

fn_write_real_data := hFile;   //保持打开状态，下次继续写入

END_FUNCTION

// MIC7001/Application/parameters/FB_PARA_DINT
FUNCTION_BLOCK FB_PARA_DINT
VAR_INPUT
	enable:BOOL := FALSE;
	clear:BOOL := FALSE;
	pPara:POINTER TO DUT_PARA_DINT;
END_VAR

VAR_OUTPUT
	ok:BOOL := FALSE;
	zero:BOOL := FALSE;
END_VAR

VAR
	hFile: RTS_IEC_HANDLE := 0;
	sync:BOOL := FALSE;  
	stat:UINT:= 0;
	
	i :UINT;
END_VAR


IF NOT enable OR pPara^.num < 1 THEN
	stat := 0;
	RETURN;
END_IF

CASE stat OF
	0:  //init
		IF rd_all(pPara^.filename)	THEN 
			zero := FALSE;
			ok := TRUE;
			stat := 10;
		ELSE
			clear_all();
			IF wr_all(pPara^.filename) THEN
				zero := TRUE;
				ok := FALSE;
				stat := 10;
			END_IF
		END_IF
	
	10: // normal
		IF chk_chg() THEN
			ok := FALSE;
			IF wr_all(pPara^.filename) THEN
				ok := TRUE;
				zero := FALSE;
			END_IF
		END_IF	
		
		IF clear THEN
			clear_all();
			IF wr_all(pPara^.filename) THEN
				zero := TRUE;
				ok := FALSE;
			END_IF
		END_IF
END_CASE

METHOD clear_all : bool
VAR_INPUT
	
END_VAR
FOR i := 1 TO pPara^.num DO
	pPara^.para[i] := 0;
	pPara^.old_val[i] := 0;
END_FOR

clear_all := TRUE;
END_METHOD

METHOD rd_all : bool
VAR_INPUT
	filename:STRING(256);
END_VAR

VAR
	iNumber:INT;
	udiByteRead:LWORD;
	udiPos:UDINT;
	udiOpenError: RTS_IEC_RESULT;
	udiReadError: RTS_IEC_RESULT;
	str: STRING(255);
	ulOffset:DWORD;
	batch: BOOL;
	check_sum: DINT;
END_VAR
rd_all := FALSE;

hFile := sysfileopen(szFile := filename, am := sysfile.AM_READ, pResult:= ADR(udiOpenError));
IF hFile = RTS_INVALID_HANDLE THEN
	RETURN;
END_IF

ulOffset := 0;
batch := TRUE;

check_sum := 0;
FOR i := 1 TO pPara^.num DO
	IF udiByteRead < 50 AND batch THEN
		udiPos := SysFileSetPos(hFile:=hFile, ulOffset := ulOffset);
		udiByteRead := sysfile.SysFileRead(hfile := hFile,pbyBuffer := ADR(str), ulSize := 255 , pResult := ADR(udiReadError));
		IF udiByteRead < 255 THEN
			batch := FALSE;
		END_IF
	END_IF
	IF udiByteRead < 1 THEN  //读取失败
		sysfile.SysFileClose(hFile := hFile);
		RETURN;
	END_IF

	iNumber := find(str, '$N');
	IF iNumber < 2 THEN
		sysfile.SysFileClose(hFile := hFile);
		RETURN;
	END_IF
	
	pPara^.para[i] := STRING_TO_DINT(left(str,iNumber-1));
	str := delete(str, iNumber,1);
	pPara^.old_val[i] := pPara^.para[i];
	
	udiByteRead := udiByteRead - ANY_TO_LWORD(iNumber);
	ulOffset := ulOffset + ANY_TO_DWORD(iNumber);

	IF i = pPara^.num THEN
		IF check_sum <> pPara^.para[i] THEN
			RETURN;  //error
		END_IF
	ELSE
		check_sum := check_sum + pPara^.para[i];
	END_IF
END_FOR

sysfile.SysFileClose(hFile := hFile);
rd_all := TRUE;
END_METHOD

METHOD chk_chg : bool
VAR_INPUT
END_VAR

VAR
	i :UINT;
END_VAR
chk_chg := TRUE;

FOR i := 1 TO pPara^.num  DO
	IF pPara^.para[i] <> pPara^.old_val[i] THEN
		RETURN;
	END_IF
END_FOR

chk_chg := FALSE;
END_METHOD

METHOD wr_all : bool
VAR_INPUT
	filename:STRING(256);
END_VAR

VAR
	iNumber:INT;
	udiByteWrite:LWORD;
	udiPos:UDINT;
	udiOpenError: RTS_IEC_RESULT;
	udiWriteError: RTS_IEC_RESULT;
	str_size:DWORD;
	str: STRING(255);
	check_sum: DINT;
END_VAR
wr_all := FALSE;
hFile := sysfileopen(szFile := filename, am := sysfile.AM_WRITE, pResult := ADR(udiOpenError));
IF hFile = RTS_INVALID_HANDLE THEN
	RETURN;
END_IF

udiPos := SysFileSetPos(hFile:=hFile, ulOffset := 0);

check_sum := 0;
str:= ANY_TO_STRING('');
FOR i := 1 TO pPara^.num DO
	IF i = pPara^.num THEN  //the last val, check_sum
		pPara^.para[i] := check_sum;
	ELSE
		check_sum := check_sum + pPara^.para[i];
	END_IF
	str := concat(str, ANY_TO_STRING(pPara^.para[i]));
	str := concat(str, ANY_TO_STRING('$N'));
	str_size := ANY_TO_DWORD(len(str));
	IF str_size > 200 THEN
		udiByteWrite := sysfile.SysFileWrite(hFile := hFile,pbyBuffer := ADR(str),ulSize := str_size, pResult := ADR(udiWriteError));
		IF udiByteWrite = str_size THEN
			str := '';
		END_IF
	END_IF	
END_FOR
udiByteWrite := sysfile.SysFileWrite(hFile := hFile,pbyBuffer := ADR(str),ulSize := str_size, pResult := ADR(udiWriteError));
	
IF udiByteWrite <> str_size THEN
	sysfile.SysFileClose(hFile);
	RETURN;
END_IF
sysfile.SysFileClose(hFile);

	
FOR i := 1 TO pPara^.num DO
	pPara^.old_val[i] := pPara^.para[i];
END_FOR

hFile := 0;

wr_all := TRUE;
END_METHOD

END_FUNCTION_BLOCK

// MIC7001/Application/prg_can0
PROGRAM prg_can0
VAR
	CAN0: CAN.CANDriver_29bit;
	mid_can_cntr:DINT:=0;
	
	tTimeLimit		: TIME := T#5MS;
	diagnosis		: CAN.CANBusDiagnosis;
	
	msgf003:MsgProcessor_j1939_f003;
	msgf004:MsgProcessor_j1939_f004;
	msgfeee: MsgProcessor_j1939_feee;
	msgfeef: MsgProcessor_j1939_feef;
	msgfef2:MsgProcessor_j1939_fef2;
	msgmid: MsgProcessor_MID;
	
	Receiver_f003: CAN.CANSingleIdReceiver;
	Receiver_f004: CAN.CANSingleIdReceiver;
	Receiver_fef2: CAN.CANSingleIdReceiver;
	Receiver_feee: CAN.CANSingleIdReceiver;
	Receiver_feef: CAN.CANSingleIdReceiver;

	Receiver_MID: CAN.CANAreaReceiver;
	
	can0_sender: CAN.CANSender;
	Message_send : CAN.RxMESSAGE;
	xSendCmd:BOOL := FALSE;
	xita: REAL;
	
	send_id:UDINT := 16#501;
	
	cntr_grade: INT;
	bData: BYTE;

	dt_send: DATE_AND_TIME;
	get_dt:dtu.GetDateAndTime;
	uiYear: UINT;
	uiMonth: UINT;
	uiDay: UINT;
	uiHour: UINT;
	uiMinute: UINT;
	uiSecond: UINT;	
	send_data_ok: BOOL := FALSE;
	can0_busy_cntr:DINT:=0;
END_VAR

VAR_INPUT	
	dtu_set_dt_fb: dtu.SetDateAndTime;
END_VAR
VAR // added by the converter: edge detectors and wires of the graphical bodies
    _s1 : CAN.DRIVER_CONFIG;
    _s2 : CAN.DIAGNOSIS_INFO;
    _s3, _s4, _s5, _s6, _s8 : CAN.RECEIVER_SINGLE_ID;
    _s7 : can.RECEIVER_AREA;
END_VAR

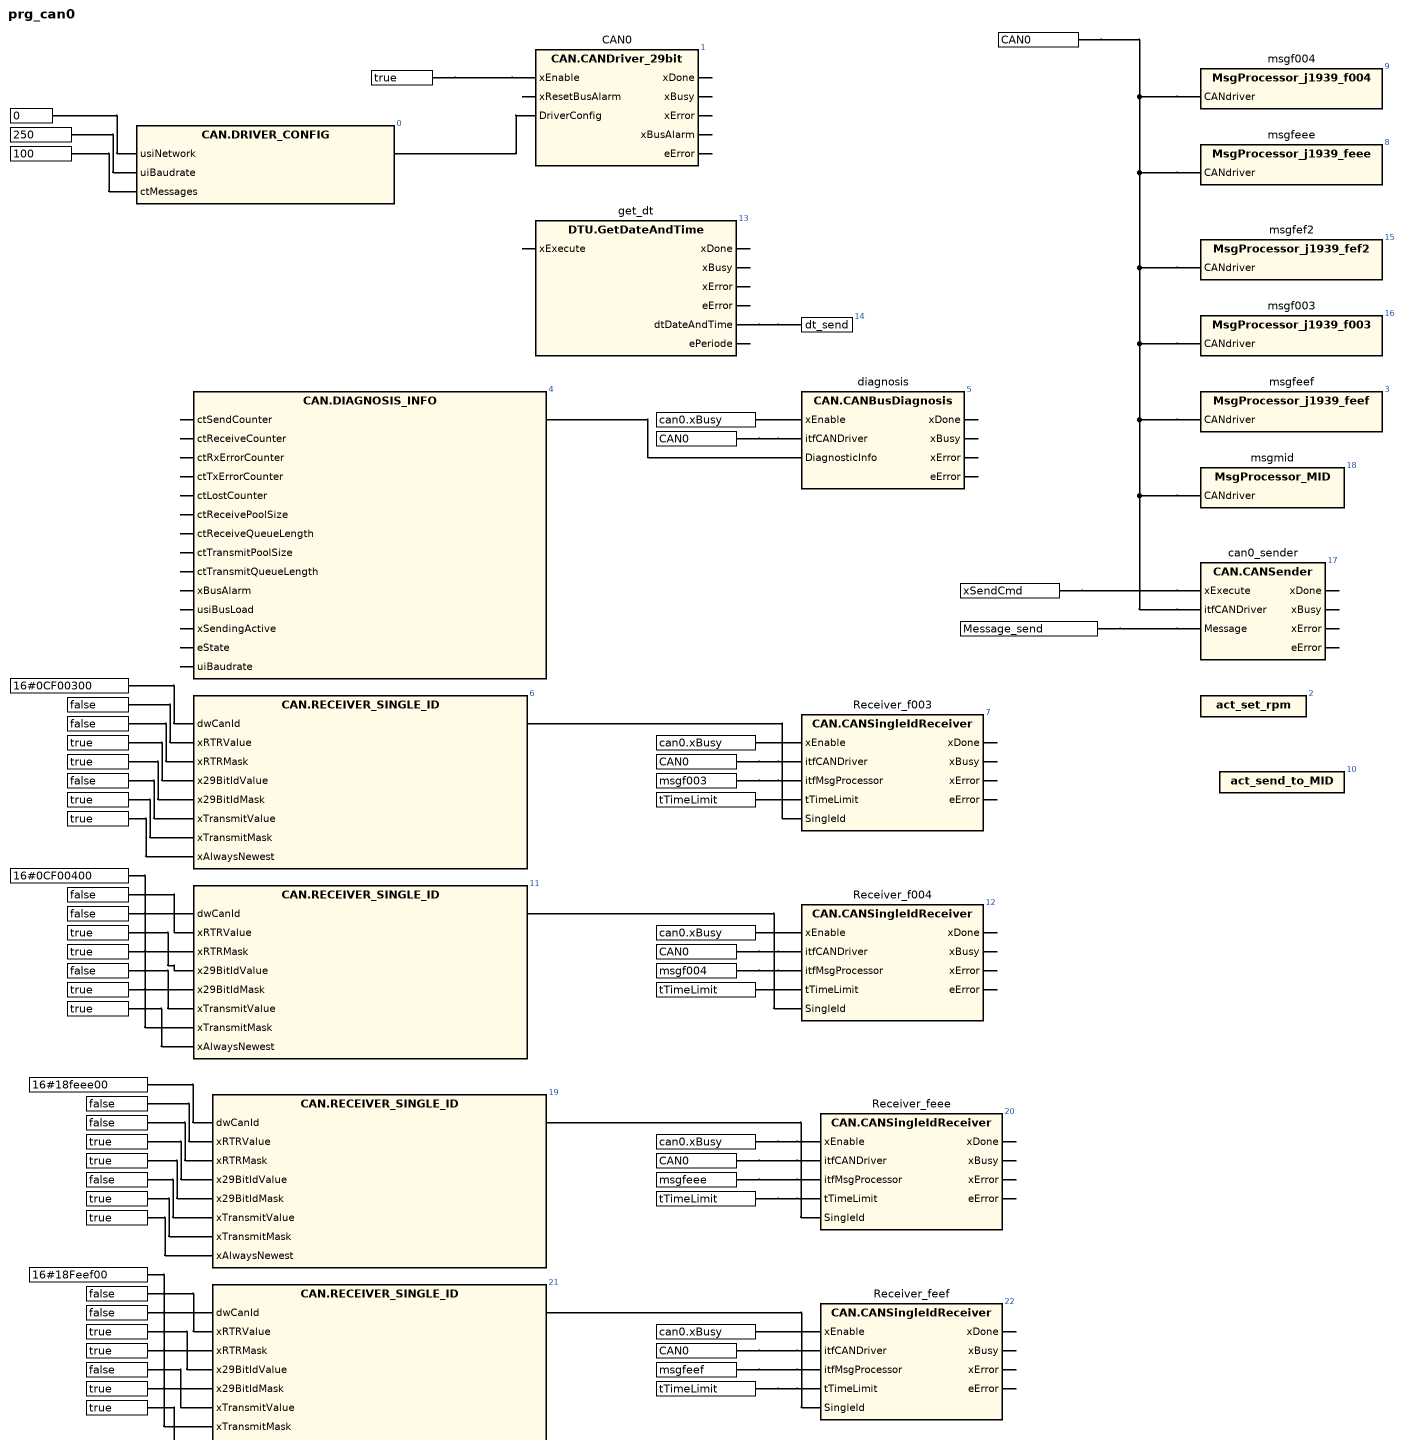
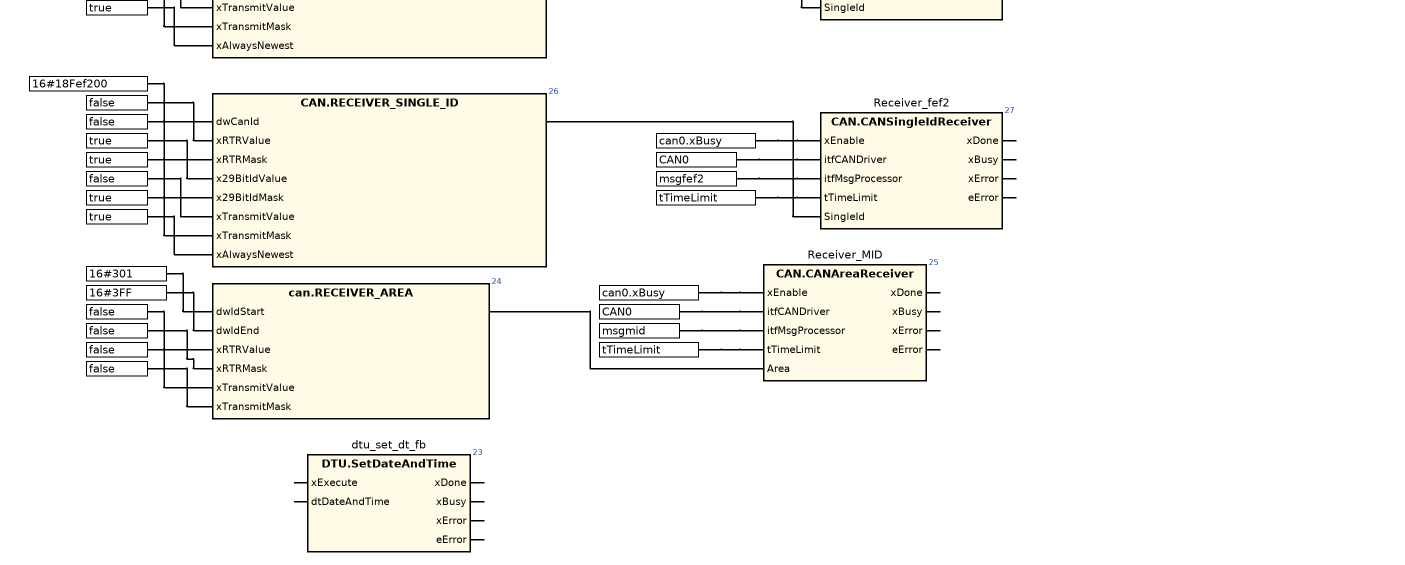
// compose _s1 : CAN.DRIVER_CONFIG
_s1.usiNetwork := 0;
_s1.uiBaudrate := 250;
_s1.ctMessages := 100;
CAN0(xEnable := true, DriverConfig := _s1); // CAN.CANDriver_29bit
act_set_rpm();
msgfeef(CANdriver := CAN0); // MsgProcessor_j1939_feef
// compose _s2 : CAN.DIAGNOSIS_INFO
diagnosis(xEnable := can0.xBusy, itfCANDriver := CAN0, DiagnosticInfo := _s2); // CAN.CANBusDiagnosis
// compose _s3 : CAN.RECEIVER_SINGLE_ID
_s3.dwCanId := 16#0CF00300;
_s3.xRTRValue := false;
_s3.xRTRMask := false;
_s3.x29BitIdValue := true;
_s3.x29BitIdMask := true;
_s3.xTransmitValue := false;
_s3.xTransmitMask := true;
_s3.xAlwaysNewest := true;
Receiver_f003(
    xEnable := can0.xBusy,
    itfCANDriver := CAN0,
    itfMsgProcessor := msgf003,
    tTimeLimit := tTimeLimit,
    SingleId := _s3); // CAN.CANSingleIdReceiver
msgfeee(CANdriver := CAN0); // MsgProcessor_j1939_feee
msgf004(CANdriver := CAN0); // MsgProcessor_j1939_f004
act_send_to_MID();
// compose _s4 : CAN.RECEIVER_SINGLE_ID
_s4.dwCanId := 16#0CF00400;
_s4.xRTRValue := false;
_s4.xRTRMask := false;
_s4.x29BitIdValue := true;
_s4.x29BitIdMask := true;
_s4.xTransmitValue := false;
_s4.xTransmitMask := true;
_s4.xAlwaysNewest := true;
Receiver_f004(
    xEnable := can0.xBusy,
    itfCANDriver := CAN0,
    itfMsgProcessor := msgf004,
    tTimeLimit := tTimeLimit,
    SingleId := _s4); // CAN.CANSingleIdReceiver
get_dt(); // DTU.GetDateAndTime
dt_send := get_dt.dtDateAndTime;
msgfef2(CANdriver := CAN0); // MsgProcessor_j1939_fef2
msgf003(CANdriver := CAN0); // MsgProcessor_j1939_f003
can0_sender(xExecute := xSendCmd, itfCANDriver := CAN0, Message := Message_send); // CAN.CANSender
msgmid(CANdriver := CAN0); // MsgProcessor_MID
// compose _s5 : CAN.RECEIVER_SINGLE_ID
_s5.dwCanId := 16#18feee00;
_s5.xRTRValue := false;
_s5.xRTRMask := false;
_s5.x29BitIdValue := true;
_s5.x29BitIdMask := true;
_s5.xTransmitValue := false;
_s5.xTransmitMask := true;
_s5.xAlwaysNewest := true;
Receiver_feee(
    xEnable := can0.xBusy,
    itfCANDriver := CAN0,
    itfMsgProcessor := msgfeee,
    tTimeLimit := tTimeLimit,
    SingleId := _s5); // CAN.CANSingleIdReceiver
// compose _s6 : CAN.RECEIVER_SINGLE_ID
_s6.dwCanId := 16#18Feef00;
_s6.xRTRValue := false;
_s6.xRTRMask := false;
_s6.x29BitIdValue := true;
_s6.x29BitIdMask := true;
_s6.xTransmitValue := false;
_s6.xTransmitMask := true;
_s6.xAlwaysNewest := true;
Receiver_feef(
    xEnable := can0.xBusy,
    itfCANDriver := CAN0,
    itfMsgProcessor := msgfeef,
    tTimeLimit := tTimeLimit,
    SingleId := _s6); // CAN.CANSingleIdReceiver
dtu_set_dt_fb(); // DTU.SetDateAndTime
// compose _s7 : can.RECEIVER_AREA
_s7.dwIdStart := 16#301;
_s7.dwIdEnd := 16#3FF;
_s7.xRTRValue := false;
_s7.xRTRMask := false;
_s7.xTransmitValue := false;
_s7.xTransmitMask := false;
Receiver_MID(
    xEnable := can0.xBusy,
    itfCANDriver := CAN0,
    itfMsgProcessor := msgmid,
    tTimeLimit := tTimeLimit,
    Area := _s7); // CAN.CANAreaReceiver
// compose _s8 : CAN.RECEIVER_SINGLE_ID
_s8.dwCanId := 16#18Fef200;
_s8.xRTRValue := false;
_s8.xRTRMask := false;
_s8.x29BitIdValue := true;
_s8.x29BitIdMask := true;
_s8.xTransmitValue := false;
_s8.xTransmitMask := true;
_s8.xAlwaysNewest := true;
Receiver_fef2(
    xEnable := can0.xBusy,
    itfCANDriver := CAN0,
    itfMsgProcessor := msgfef2,
    tTimeLimit := tTimeLimit,
    SingleId := _s8); // CAN.CANSingleIdReceiver

ACTION act_set_rpm:

IF NOT CAN0.xBusy THEN
	RETURN;
END_IF

IF can0_sender.xBusy THEN
	RETURN;
END_IF

IF can0_sender.xError THEN
	can0_sender(xExecute := FALSE, Message := Message_send);
END_IF 

IF can0_sender.xDone THEN
	can0_sender(xExecute := FALSE, Message := Message_send);
END_IF

IF can0_sender.xExecute THEN
	can0_sender(xExecute := FALSE, Message := Message_send);
END_IF

Message_send.abyData[0] := 16#31;
Message_send.abyData[1] := DINT_TO_BYTE(gvl.g_rpm_set*8 MOD 256);;
Message_send.abyData[2] := DINT_TO_BYTE(gvl.g_rpm_set*8 / 256);;
Message_send.abyData[3] := 0;
Message_send.abyData[4] := 0;
Message_send.abyData[5] := 0;
Message_send.abyData[6] := 16#FF;
Message_send.abyData[7] := 16#FF;

Message_send.udiCanID := 16#C000007;
Message_send.usiDataLength := 8;
Message_send.xIs29BitMessage := TRUE;
Message_send.xIsTxMessage := TRUE;
Message_send.xRTR := FALSE;

xSendCmd := TRUE;  //send

RETURN;
END_ACTION

ACTION act_send_to_MID:
IF mid_can_cntr < 10 THEN
	mid_can_cntr := mid_can_cntr + 1;
	RETURN;
END_IF
mid_can_cntr := 0;

IF NOT CAN0.xBusy THEN
	can0_busy_cntr := can0_busy_cntr+1;
	RETURN;
END_IF
can0_busy_cntr := 0;

IF can0_sender.xBusy THEN
	RETURN;
END_IF

IF can0_sender.xError THEN
	can0_sender(xExecute := FALSE, Message := Message_send);
END_IF 

IF can0_sender.xDone THEN
	can0_sender(xExecute := FALSE, Message := Message_send);
END_IF

//填充并发送到显示屏的数据，每个周期发送一帧
// from 16#501  --->  16#506
send_data_ok := FALSE;

CASE send_id OF
16#501:

	bData := 0;
	bData.2 := gvl.cmd_auto_idle;
	bData.3 := gvl.cmd_high_speed;
	bData.4 := gvl.cmd_more_power;
	bData.5 := gvl.cmd_clear_hours;
	bData.6 := gvl.cmd_clear_hours_1;
	bData.7 := gvl.cmd_clear_hours_2;
	Message_send.abyData[0] := bData;
	Message_send.abyData[1] := ANY_TO_BYTE(gvl.g_ai_fuel_level);
	Message_send.abyData[2] := ANY_TO_BYTE(gvl.g_temp_coolant_1939);
	Message_send.abyData[3] := ANY_TO_BYTE(gvl.ai_vcc/100 - 100);
	Message_send.abyData[4] := ANY_TO_BYTE(gvl.g_rpm_real);
	Message_send.abyData[5] := ANY_TO_BYTE(gvl.g_rpm_real/256);
	Message_send.abyData[6] := ANY_TO_BYTE(gvl.g_res_prop);
	Message_send.abyData[7] := 0;
	send_data_ok := TRUE;

16#502:

	Message_send.abyData[0] := ANY_TO_BYTE(gvl.gear_grade);
	Message_send.abyData[1] := ANY_TO_BYTE(g_Eng_Oil_Temp+40);
	Message_send.abyData[2] := ANY_TO_BYTE(gvl.g_load_percent_1939);
	
	bData := 0;
	bData.0 := (g_oil_press_1939 < 100);
	bData.1 := FALSE; //液压油污
	bData.2 := FALSE; //备用
	bData.3 := FALSE; //机械怠速
	bData.4 := FALSE; //空滤阻塞
	bData.5 := (gvl.g_rpm_real < 500); //电池放电
	bData.6 := FALSE; //先导油滤
	bData.7 := (g_temp_coolant_1939 > 98); //水温开关量
	Message_send.abyData[3] := bData;
	
	bData := 0;
	
	Message_send.abyData[4] := 0;
	Message_send.abyData[5] := 0;
	Message_send.abyData[6] := 0;
	Message_send.abyData[7] := 0;
	send_data_ok := TRUE;

16#503:
	bData := ANY_TO_BYTE(gvl.g_ai_curr_prop MOD 256);
	Message_send.abyData[0] := bData;
	
	bData := ANY_TO_BYTE(gvl.g_ai_curr_prop/256);
	Message_send.abyData[1] := bData;
	
	bData := ANY_TO_BYTE(ANY_TO_DINT(gvl.g_ai_pilot*1000.0) MOD 256);
	Message_send.abyData[2] := bData;
	
	bData := ANY_TO_BYTE(ANY_TO_DINT(gvl.g_ai_pilot*1000.0)/256);
	Message_send.abyData[3] := bData;

	bData := ANY_TO_BYTE(ANY_TO_DINT(gvl.g_ai_press_pump1*1000.0) MOD 256);
	Message_send.abyData[4] := bData;
	
	bData := ANY_TO_BYTE(ANY_TO_DINT(gvl.g_ai_press_pump1*1000.0)/256);
	Message_send.abyData[5] := bData;

	bData := ANY_TO_BYTE(ANY_TO_DINT(gvl.g_ai_press_pump2*1000.0) MOD 256);
	Message_send.abyData[6] := bData;
	
	bData := ANY_TO_BYTE(ANY_TO_DINT(gvl.g_ai_press_pump2*1000.0)/256);
	Message_send.abyData[7] := bData;	
	send_data_ok := TRUE;

16#504:
	bData := ANY_TO_BYTE(gvl.g_machine_mins MOD 256);
	Message_send.abyData[0] := bData;
	
	bData := ANY_TO_BYTE(gvl.g_machine_mins/256 MOD 256);
	Message_send.abyData[1] := bData;
	
	bData := ANY_TO_BYTE(gvl.g_machine_mins/256/256 MOD 256);
	Message_send.abyData[2] := bData;
	
	bData := ANY_TO_BYTE(gvl.g_machine_mins/256/256/256);
	Message_send.abyData[3] := bData;
	
	bData := ANY_TO_BYTE(gvl.g_machine_mins_1 MOD 256);
	Message_send.abyData[4] := bData;

	bData := ANY_TO_BYTE(gvl.g_machine_mins_1/256);
	Message_send.abyData[5] := bData;	

	bData := ANY_TO_BYTE(gvl.g_machine_mins_2 MOD 256);
	Message_send.abyData[6] := bData;

	bData := ANY_TO_BYTE(gvl.g_machine_mins_2/256);
	Message_send.abyData[7] := bData;		
	send_data_ok := TRUE;
	
16#505:  //油耗相关数据
	Message_send.abyData[0] := ANY_TO_BYTE(ANY_TO_UINT(gvl.g_fuel_rate_1939) MOD 256);
	Message_send.abyData[1] := ANY_TO_BYTE(ANY_TO_UINT(gvl.g_fuel_rate_1939) / 256);

	Message_send.abyData[2] := ANY_TO_BYTE(ANY_TO_UINT(gvl.g_fuel_depleted/100) MOD 256);
	Message_send.abyData[3] := ANY_TO_BYTE(ANY_TO_UINT(gvl.g_fuel_depleted/100) / 256);

	Message_send.abyData[4] := ANY_TO_BYTE(ANY_TO_UINT(gvl.g_fuel_depleted_1) MOD 256);
	Message_send.abyData[5] := ANY_TO_BYTE(ANY_TO_UINT(gvl.g_fuel_depleted_1) / 256);

	Message_send.abyData[6] := ANY_TO_BYTE(ANY_TO_UINT(gvl.g_fuel_depleted_2) MOD 256);
	Message_send.abyData[7] := ANY_TO_BYTE(ANY_TO_UINT(gvl.g_fuel_depleted_2) / 256);
	send_data_ok := TRUE;
	
	get_dt.xExecute := TRUE;  //读取系统时间，为506做准备
	
16#506:
	IF uiYear < 2000 THEN   //错误的时间一般为1970年
		gvl.g_time_good := FALSE;
	ELSE
		Message_send.abyData[0] := ANY_TO_BYTE(uiSecond);
		Message_send.abyData[1] := ANY_TO_BYTE(uiMinute);
		Message_send.abyData[2] := ANY_TO_BYTE(uiHour);
		Message_send.abyData[3] := ANY_TO_BYTE(uiDay);
		Message_send.abyData[4] := ANY_TO_BYTE(uiMonth);
		Message_send.abyData[5] := ANY_TO_BYTE(uiYear-2000);
		gvl.g_time_good := TRUE;
		Message_send.abyData[6] := 0;
		Message_send.abyData[7] := ANY_TO_BYTE(gvl.g_time_good);
		send_data_ok := TRUE;
	END_IF
	
END_CASE

IF get_dt.xDone THEN
	uiYear := 0;
	dtu.DTSplit(dt_send, ADR(uiYear), ADR(uiMonth), ADR(uiDay), ADR(uiHour), ADR(uiMinute), ADR(uiSecond));
	get_dt(xExecute := FALSE);
END_IF

IF send_data_ok THEN
	Message_send.udiCanID := send_id;
	Message_send.usiDataLength := 8;
	Message_send.xIs29BitMessage := FALSE;
	Message_send.xIsTxMessage := TRUE;
	Message_send.xRTR := FALSE;
	xSendCmd := TRUE;  //send
END_IF

send_id := send_id+1;
IF send_id > 16#506 THEN
	send_id := 16#501;	
END_IF

RETURN;
END_ACTION

END_PROGRAM

// MIC7001/Application/function_blocks/MsgProcessor_j1939_feef
/// MsgProcessor_Echo is the implimentation of IMessageProcessor. 
/// MsgProcessor_Echo simply counts all incoming messages and echos them with CobId +1
FUNCTION_BLOCK MsgProcessor_j1939_feef IMPLEMENTS CAN.IMessageProcessor
VAR_IN_OUT
	CANdriver	: CAN.CANdriver_29bit;
END_VAR
VAR_OUTPUT
END_VAR
VAR
	_pCANdriver : POINTER TO CAN.CANdriver_29bit;
END_VAR

_pCANdriver := ADR(CANdriver);

METHOD ProcessMessage
VAR_IN_OUT
	(* The messages received by the receiver *)
	Message	: CAN.RxMessage;
END_VAR
VAR
END_VAR
IF _pCANdriver = 0 THEN
	RETURN;
END_IF

gvl.g_oil_press_1939 := ANY_TO_REAL(Message.abyData[3])*4.0;   //0~1000 KPa
gvl.g_coolant_level_1939 := ANY_TO_REAL(Message.abyData[7])*0.4;  //0~100%
END_METHOD

END_FUNCTION_BLOCK

// MIC7001/Application/function_blocks/MsgProcessor_j1939_feee
/// MsgProcessor_Echo is the implimentation of IMessageProcessor. 
/// MsgProcessor_Echo simply counts all incoming messages and echos them with CobId +1
FUNCTION_BLOCK MsgProcessor_j1939_feee IMPLEMENTS CAN.IMessageProcessor
VAR_IN_OUT
	CANdriver	: CAN.CANdriver_29bit;
END_VAR
VAR_OUTPUT
END_VAR
VAR
	_pCANdriver : POINTER TO CAN.CANdriver_29bit;
END_VAR

_pCANdriver := ADR(CANdriver);

METHOD ProcessMessage
VAR_IN_OUT
	(* The messages received by the receiver *)
	Message	: CAN.RxMessage;
END_VAR
VAR
END_VAR
IF _pCANdriver = 0 THEN
	RETURN;
END_IF

gvl.g_temp_coolant_1939:=temp_neg40_to_210oC(Message.abyData[0]);
gvl.g_Eng_Fuel_Temp:=temp_neg40_to_210oC(Message.abyData[1]);
gvl.g_Eng_Oil_Temp:=temp_absZero_to_1735oC(Message.abyData[2]+Message.abyData[3]*16#100);
gvl.g_Turbo_Oil_Temp:=temp_absZero_to_1735oC(Message.abyData[4]+Message.abyData[5]*16#100);
gvl.g_Eng_InterCooler_Temp:=temp_neg40_to_210oC(Message.abyData[6]);
gvl.g_Eng_InterCooler_Thermostat_Opening:=pros100(Message.abyData[7]);
END_METHOD

END_FUNCTION_BLOCK

// MIC7001/Application/j1939/temp_neg40_to_210oC
FUNCTION temp_neg40_to_210oC : INT
VAR_INPUT
	data:USINT;
END_VAR
VAR
END_VAR

temp_neg40_to_210oC := ANY_TO_INT(data) - 40;

END_FUNCTION

// MIC7001/Application/j1939/temp_absZero_to_1735oC
FUNCTION temp_absZero_to_1735oC : INT
VAR_INPUT
	data:UINT;
END_VAR
VAR
END_VAR

temp_absZero_to_1735oC := ANY_TO_INT(data/32)-273;

END_FUNCTION

// MIC7001/Application/j1939/pros100
FUNCTION pros100 : USINT
VAR_INPUT
	data :USINT;
END_VAR
VAR
	d:UINT;
END_VAR

d := data*4/10;
IF d > 100 THEN
	d := 100;
END_IF

pros100 := ANY_TO_USINT(d);

END_FUNCTION

// MIC7001/Application/function_blocks/MsgProcessor_j1939_f004
/// MsgProcessor_Echo is the implimentation of IMessageProcessor. 
/// MsgProcessor_Echo simply counts all incoming messages and echos them with CobId +1
FUNCTION_BLOCK MsgProcessor_j1939_f004 IMPLEMENTS CAN.IMessageProcessor
VAR_IN_OUT
	CANdriver	: CAN.CANdriver_29bit;
END_VAR
VAR_OUTPUT
END_VAR
VAR
	_pCANdriver : POINTER TO CAN.CANdriver_29bit;
END_VAR

_pCANdriver := ADR(CANdriver);

METHOD ProcessMessage
VAR_IN_OUT
	(* The messages received by the receiver *)
	Message	: CAN.RxMessage;
END_VAR
VAR
END_VAR
IF _pCANdriver = 0 THEN
	RETURN;
END_IF

gvl.g_rpm_real := (Message.abyData[3] + Message.abyData[4]*256)/8;

gvl.g_demand_torque_1939 := ANY_TO_REAL(Message.abyData[1]) - 125.0;

gvl.g_real_torque_1939 := ANY_TO_REAL(Message.abyData[2]) - 125.0;
END_METHOD

END_FUNCTION_BLOCK

// MIC7001/Application/function_blocks/MsgProcessor_j1939_fef2
/// MsgProcessor_Echo is the implimentation of IMessageProcessor. 
/// MsgProcessor_Echo simply counts all incoming messages and echos them with CobId +1
FUNCTION_BLOCK MsgProcessor_j1939_fef2 IMPLEMENTS CAN.IMessageProcessor
VAR_IN_OUT
	CANdriver	: CAN.CANdriver_29bit;
END_VAR
VAR_OUTPUT
END_VAR
VAR
	_pCANdriver : POINTER TO CAN.CANdriver_29bit;
END_VAR

_pCANdriver := ADR(CANdriver);

METHOD ProcessMessage
VAR_IN_OUT
	(* The messages received by the receiver *)
	Message	: CAN.RxMessage;
END_VAR
VAR
END_VAR
IF _pCANdriver = 0 THEN
	RETURN;
END_IF

//计算瞬时油耗， 单位: 毫升/秒
gvl.g_fuel_rate_1939 := ANY_TO_REAL(Message.abyData[1]*256 + Message.abyData[0])*1000.0/20.0/3600.0;
END_METHOD

END_FUNCTION_BLOCK

// MIC7001/Application/function_blocks/MsgProcessor_j1939_f003
/// MsgProcessor_Echo is the implimentation of IMessageProcessor. 
/// MsgProcessor_Echo simply counts all incoming messages and echos them with CobId +1
FUNCTION_BLOCK MsgProcessor_j1939_f003 IMPLEMENTS CAN.IMessageProcessor
VAR_IN_OUT
	CANdriver	: CAN.CANdriver_29bit;
END_VAR
VAR_OUTPUT
END_VAR
VAR
	_pCANdriver : POINTER TO CAN.CANdriver_29bit;
END_VAR

_pCANdriver := ADR(CANdriver);

METHOD ProcessMessage
VAR_IN_OUT
	(* The messages received by the receiver *)
	Message	: CAN.RxMessage;
END_VAR
VAR
END_VAR
IF _pCANdriver = 0 THEN
	RETURN;
END_IF

gvl.g_load_percent_1939 := ANY_TO_REAL(Message.abyData[2]);
END_METHOD

END_FUNCTION_BLOCK

// MIC7001/Application/function_blocks/MsgProcessor_MID
/// MsgProcessor_Echo is the implimentation of IMessageProcessor. 
/// MsgProcessor_Echo simply counts all incoming messages and echos them with CobId +1
FUNCTION_BLOCK MsgProcessor_MID IMPLEMENTS CAN.IMessageProcessor
VAR_IN_OUT
	CANdriver	: CAN.CANdriver_29bit;
END_VAR
VAR_OUTPUT
END_VAR
VAR
	_pCANdriver : POINTER TO CAN.CANdriver_29bit;
	r_triger_mins:r_trig;
	r_triger_mins_1:r_trig;
	r_triger_mins_2:r_trig;
	
END_VAR

_pCANdriver := ADR(CANdriver);

METHOD ProcessMessage
VAR_IN_OUT
	(* The messages received by the receiver *)
	Message	: CAN.RxMessage;
END_VAR
VAR
	bData: BYTE;
	new_dt : DATE_AND_TIME;
	
	bTime_min: BYTE;
	bTime_sec: BYTE;
	bTime_hour: BYTE;
	bTime_date: BYTE;
	bTime_month: BYTE;
	bTime_year: BYTE;
	bTime_week: BYTE;
	bTime_good: BYTE;
	str_dt: STRING(255);
END_VAR
IF _pCANdriver = 0 THEN
	RETURN;
END_IF

CASE Message.udiCanID OF
16#301:
	bData := Message.abyData[0];
	gvl.g_mode := ANY_TO_BYTE(bData.0) + ANY_TO_BYTE(bData.1)*2;
	gvl.cmd_auto_idle  := bData.2;
	gvl.cmd_high_speed := bData.3;
	gvl.cmd_more_power := bData.4;
	
	gvl.cmd_clear_hours := bData.5;
	gvl.cmd_clear_hours_1 := bData.6;
	gvl.cmd_clear_hours_2 := bData.7;
	
	r_triger_mins(clk := bData.5);
	IF r_triger_mins.Q AND gvl.g_machine_mins < 20*60  THEN  //清空小时计, 只有在小于20小时的情况下允许
		gvl.g_machine_start_mins := gvl.g_running_mins;
		prg_data.para_dint.para[35] := gvl.g_running_mins;
		gvl.g_machine_mins := gvl.g_running_mins - gvl.g_machine_start_mins;
	END_IF

	r_triger_mins_1(clk := bData.6);
	IF r_triger_mins_1.Q THEN  //清空阶段一小时计
		gvl.g_machine_mins_1_start := gvl.g_running_mins;
	END_IF

	r_triger_mins_2(clk := bData.7);
	IF r_triger_mins_2.Q THEN  //清空阶段二小时计
		gvl.g_machine_mins_2_start := gvl.g_running_mins;
	END_IF	
	
16#302:
	bTime_sec := Message.abyData[0];
	bTime_min := Message.abyData[1];
	bTime_hour := Message.abyData[2];
	bTime_date := Message.abyData[3];
	bTime_month := Message.abyData[4];
	bTime_year := Message.abyData[5];
	bTime_week := Message.abyData[6];
	bTime_good := Message.abyData[7];
	
	IF bTime_good > 0 AND NOT gvl.g_time_good THEN
		str_dt := concat('dt#', ANY_TO_STRING(2000+bTime_year));
		str_dt := concat(str_dt, '-');
		str_dt := concat(str_dt, ANY_TO_STRING(bTime_month));
		str_dt := concat(str_dt, '-');
		str_dt := concat(str_dt, ANY_TO_STRING(bTime_date));
		str_dt := concat(str_dt, '-');
		str_dt := concat(str_dt, ANY_TO_STRING(bTime_hour));
		str_dt := concat(str_dt, ':');
		str_dt := concat(str_dt, ANY_TO_STRING(bTime_min));
		str_dt := concat(str_dt, ':');
		str_dt := concat(str_dt, ANY_TO_STRING(bTime_sec));
		prg_can0.dtu_set_dt_fb.dtDateAndTime := STRING_TO_DT(str_dt);
		prg_can0.dtu_set_dt_fb(xExecute := FALSE);
		prg_can0.dtu_set_dt_fb.xExecute := TRUE;
		gvl.g_time_good := TRUE;
	END_IF
END_CASE
END_METHOD

END_FUNCTION_BLOCK

// MIC7001/Application/prg_set_inmode
PROGRAM prg_set_inmode
VAR
	stat:UINT := 0;
	old_in_mode:ARRAY[0..47] OF UINT;  //从已有文件中读出的配置
	in_mode:ARRAY[0..47] OF UINT;   //当前设定的配置
	number :UINT := 48;  //通道总数
	i: UINT;
END_VAR


CASE stat OF
0: //read inmode.txt
	IF fn_read_in_mode_file(pInMOde := ADR(old_in_mode), number := number) THEN
		stat := 50;
	ELSE 
		stat := 10;
	END_IF
10: //need write
	IF fn_write_in_mode_file(pInMode := ADR(in_mode), number := number) THEN
		stat := 100; //succeed
	END_IF

50: //the file inmode.txt is exist.
	FOR i := 0 TO number-1 DO
		IF old_in_mode[i] <> in_mode[i] THEN
			stat := 10; //write new config
			RETURN;
		END_IF
	END_FOR
	stat := 100;

100: //succeed, return;
	RETURN;
END_CASE

FOR  i := 0 TO number-1 DO
	in_mode[i] := 0;
END_FOR

in_mode[5] := 3;  //0~30 ohm 油水分离
in_mode[8] := 4;  //开机信号
in_mode[6] := 5;  //空滤阻塞
in_mode[7] := 4;
in_mode[28] := 3;  //油温传感器，可变电阻（原系统使用9.4V电压上拉）
in_mode[46] := 3;  //柴油 油位
in_mode[0] := 2;   //先导压力，6MPa
in_mode[24] := 5;
in_mode[25] := 4;
in_mode[26] := 4;
in_mode[27] := 4;
in_mode[1] := 2;  //前泵主压，40MPa， 内部增焊250 ohm电阻，使用0~20mA模式采集电流
in_mode[2] := 2;  //后泵主压，40MPa，内部增焊250 ohm电阻，使用0~20mA模式采集电流
in_mode[18] := 1;
in_mode[19] := 1;
in_mode[20] := 1;
in_mode[21] := 1;
in_mode[22] := 1;
in_mode[23] := 1;

END_PROGRAM

// MIC7001/Application/functions/fn_read_in_mode_file
FUNCTION fn_read_in_mode_file : BOOL
VAR_INPUT
	pInMode :POINTER TO UINT;
	number:UINT;
END_VAR
VAR
	hFile: RTS_IEC_HANDLE;
	udiOpenError: RTS_IEC_RESULT;
	udiReadError: RTS_IEC_RESULT;
	i :DWORD;
	iTemp: UDINT;
	udiPos: UDINT;
	str: STRING(65535);
	str_size: __XWORD;
	udiByteRead: LWORD;

	len_of_line: INT;
	len_of_number :INT;
	magicNumber:REAL;
	check_sum:REAL:= 0;
	temp_num:REAL;
	index :UINT;
	mode: UINT;
END_VAR

fn_read_in_mode_file := FALSE;

//检测文件是否存在
hFile := sysfileopen(szFile := gvl.inmode_file, am := sysfile.AM_READ, pResult:= ADR(udiOpenError));
IF hFile = RTS_INVALID_HANDLE	THEN  //文件不存在
	RETURN;
END_IF

//文件存在，开始读取内容
udiPos := SysFileSetPos(hFile:=hFile, ulOffset := 0);
udiByteRead := sysfile.SysFileRead(hfile := hFile,pbyBuffer := ADR(str), ulSize := SIZEOF(str), pResult := ADR(udiReadError));
IF udiByteRead < 1 THEN  //读取失败
	sysfile.SysFileClose(hFile := hFile);
	RETURN;
END_IF
sysfile.SysFileClose(hFile);

//读取本行的数字
FOR i := 0 TO number-1 DO
	len_of_number := find(str, '$N');
	mode := STRING_TO_UINT(left(str,len_of_number-1));
	str := delete(str, len_of_number,1);	
	pInMode[i] := mode;
END_FOR

fn_read_in_mode_file := TRUE;
RETURN;

END_FUNCTION

// MIC7001/Application/functions/fn_write_in_mode_file
FUNCTION fn_write_in_mode_file : BOOL
VAR_INPUT
	pInMode :POINTER TO UINT;
	number:UINT;
END_VAR
VAR
	bak_file_prefix:STRING :=ANY_TO_STRING("in_mode_bak_");
	bak_file:STRING := ANY_TO_STRING("");	
	hFile: RTS_IEC_HANDLE;
	udiDeleteError: RTS_IEC_RESULT;
	udiOpenError: RTS_IEC_RESULT;
	udiWriteError: RTS_IEC_RESULT;
	filesize: __XWORD;
	i :DWORD;
	iTemp: UDINT;
	udiPos: UDINT;
	str: STRING(256);
	str_size: __XWORD;
	udiByteWrite: LWORD;
	check_sum:REAL := 0;
END_VAR

fn_write_in_mode_file := FALSE;

IF number = 0 THEN
	RETURN;
END_IF

hFile := sysfileopen(szFile := gvl.inmode_file, am := sysfile.AM_WRITE, pResult := ADR(udiOpenError));
IF hFile = RTS_INVALID_HANDLE THEN //创建文件失败
	RETURN;
END_IF
	
udiPos := SysFileSetPos(hFile:=hFile, ulOffset:=0);	
str:= ANY_TO_STRING('');
FOR i := 0 TO number-1 DO
	str := concat(str, ANY_TO_STRING(pInMode[i]));
	str := concat(str, '$N');	
END_FOR

str_size := ANY_TO_DWORD(len(str));
udiByteWrite := sysfile.SysFileWrite(hFile := hFile,pbyBuffer := ADR(str),ulSize := str_size, pResult := ADR(udiWriteError));

sysfile.SysFileClose(hFile);
fn_write_in_mode_file := TRUE;

END_FUNCTION

// MIC7001/Application/GPRS/prg_heartbeat
PROGRAM prg_heartbeat
VAR_OUTPUT
	lock_state :INT := 0;
	unlock_state :INT := 0;
	lock_unlock_level :INT := 0;
	delay_time :INT := 0;
END_VAR

VAR
	is_inited :BOOL := FALSE;
	g_m26:fb_m26;
	udp_handle :CAA.HANDLE; 
	udp_write_fb:Udp_Write;
	udp_read_fb:Udp_Read;
	file_read_fb:File_Read;
	com_read_fb :Com_Read;


	size :CAA.SIZE;	
	Writebuffer: 			ARRAY[1..200] OF BYTE;
	Readbuffer: 			ARRAY[0..1499] OF BYTE;
	ReadbufferStr: STRING;
	atcState :INT := 0;
	
	writeUdpState :INT := 0;
	readUdpState :INT := 0;
	
	i :INT;
	count :INT := 0;
	
	rtc_fb: RTC;
	dtu_set_dt_fb: dtu.SetDateAndTime;
	
	sn_file_name :STRING := '/userapp/sn.txt';
	time_file_name :STRING := '/userapp/r_mins.txt';
	is_read :BOOL := FALSE;
	read_count :INT := 0;
	readFileState :INT := 0;
	ton_fb :TON;
	iccid_read_buffer :STRING;
	position :INT := -1;
	new_date:DT;
	get_iccid:fb_get_iccid;
	get_lac:fb_get_lac;
	iStat :UINT := 0;
	lac : STRING(4) := '0000';
	ci : STRING(4) := '0000';
	lenHearBeat:UINT;
	dataHearBeat:ARRAY[0..255] OF BYTE;
	ton_hb:ton; //heartbeat timer 
	bReturn:BOOL;
	lenLayer2:UINT;
	dataLayer2:ARRAY[0..255] OF BYTE;
	lenLayer1:UINT;
	lenRecvLayer1:UINT := 1500;
	dataLayer1:ARRAY[0..255] OF BYTE;
	bSN :ARRAY[0..9] OF BYTE;
	sub_str:STRING(8);
	num :UINT;
	lenHeartBeat: UINT;
	sn: STRING;
	work_time: UDINT;
	dataIndex :UINT := 0;
	cntr_lac:UINT := 0;
	cntr_iccid:UINT := 0;
	
	dataLayern:ARRAY[1..255] OF BYTE;
	recv_size :CAA.SIZE;
END_VAR

CASE iStat OF
0:
	g_m26(enable := TRUE, ipaddr := '47.107.240.29', port := 34567);  //共用的基础模块，只要有一个地方调用即可	
	IF g_m26.xDone THEN
		iStat := 1;
	END_IF

1:  // read iccid
	get_iccid(xExecute := FALSE);
	iStat := 2;
	cntr_iccid := 0;
	
2:
	get_iccid(xExecute := TRUE, m26_handle := g_m26.handle_m26);
	IF get_iccid.xDone THEN
		iccid_read_buffer := get_iccid.iccid;
		iStat := 10;
	END_IF
	cntr_iccid := cntr_iccid + 1;
	IF cntr_iccid > 600 THEN   // 1 min
		iStat := 1;
	END_IF
	
10: //read sn
	file_read_fb(file_name := sn_file_name);
	IF file_read_fb.isRead THEN
		sn := file_read_fb.sReadLine;
		iStat := 15;
	END_IF
	
15:
	get_lac(xExecute := FALSE);	
	iStat := 20;
	cntr_lac := 0;
	
20:
	get_lac(xExecute := TRUE, m26_handle := g_m26.handle_m26);
	IF get_lac.xDone THEN
		lac := get_lac.lac;
		ci := get_lac.ci;
		iStat := 30;
	END_IF
	cntr_lac := cntr_lac + 1;
	IF cntr_lac > 200 THEN
		iStat := 0;
	END_IF
	
30:
	file_read_fb(file_name := time_file_name);
	IF file_read_fb.isRead THEN
		work_time := STRING_TO_UDINT(file_read_fb.sReadLine);
		iStat := 100;
	END_IF
	
100:   //定时等待
	ton_fb(IN := TRUE, PT := T#10S);
	IF (ton_fb.Q) THEN
		ton_fb(IN := FALSE, PT := T#10S);
		iStat := 200;  //发送心跳
	ELSE
		iStat := 300; //发送实时数据	
	END_IF
	
200:
	bReturn := fn_cyber_heartBeat(	  //填充第三层：心跳帧
						lac_str := lac, 
						cid_str := ci, 
						ccid_str := iccid_read_buffer, 
						mins := work_time, 
						clientCode := 6,   //hengtian 95
						machineCode := 5,  //挖掘机
						pLenOut := ADR(lenHearBeat), 
						pDataOut := ADR(dataHearBeat));
	IF NOT bReturn THEN
		RETURN;
	END_IF;

	dataIndex := dataIndex + 1;
	bReturn := fn_cyber_layer2( //填充第二层，数据层
						dataType := 1,
						paraId := 0,
						dataIndex := dataIndex,
						ver := 1,
						res1 := 0,
						LenIn := lenHearBeat,
						pDataIn := ADR(dataHearBeat),
						pLenOut := ADR(lenLayer2),
						pDataOut := ADR(dataLayer2));
						
	IF NOT bReturn THEN
		RETURN;
	END_IF;

	bSN := fn_sn_str_to_byte(sn);
	bReturn := fn_cyber_layer1(    //填充第一层，设备层
						sn := ADR(bSN),
						ver := 1,
						lenIn := lenLayer2,
						pDataIn := ADR(dataLayer2),
						pLenOut := ADR(lenLayer1),
						pDataOut := ADR(dataLayer1));
	IF NOT bReturn THEN
		RETURN;
	ELSE
		udp_write_fb(xExecute := FALSE);
		iStat := 500;
	END_IF;
	
300:
	iStat := 100;
	
500:
	udp_write_fb(xExecute := TRUE, com := g_m26.handle_m26, buffer := ADR(dataLayer1), size := lenLayer1);
	IF udp_write_fb.xDone THEN
		udp_write_fb(xExecute := FALSE);
		udp_read_fb(xExecute := FALSE);
		iStat := 600; 
	END_IF
	
	IF udp_write_fb.xError THEN  
		udp_write_fb(xExecute := FALSE);
		iStat := 30; 
	END_IF
	
	
600:
	udp_read_fb(xExecute := TRUE, com := g_m26.handle_m26, buffer := ADR(Readbuffer), rsize := sizeof(Readbuffer));
	IF udp_read_fb.xDone THEN  //接收到数据
	 	recv_size := udp_read_fb.size;
		udp_read_fb(xExecute := FALSE);
		iStat := 30; //read mins and lca again
		IF recv_size = 25 THEN
			lock_state := BYTE_TO_INT(Readbuffer[20]);
			unlock_state := BYTE_TO_INT(Readbuffer[21]);
			lock_unlock_level := BYTE_TO_INT(Readbuffer[22]);
			delay_time := BYTE_TO_INT(Readbuffer[23]);
		END_IF
	END_IF
	
	IF udp_read_fb.xError THEN  //接收错误
		udp_read_fb(xExecute := FALSE);
		recv_size := 0;
		iStat := 30; //read mins and lca again
	END_IF

END_CASE

RETURN;

END_PROGRAM

// MIC7001/Application/GPRS/fn_cyber_heartBeat
FUNCTION fn_cyber_heartBeat : bool
VAR_INPUT
	lac_str:STRING(4);
	cid_str:STRING(4);
	ccid_str:STRING(21);
	mins:UDINT;
	clientCode:UINT;
	machineCode:UINT;
	pLenOut:POINTER TO UINT;
	pDataOut:POINTER TO BYTE;
END_VAR
VAR
	index: UINT;
	data_uint: UINT;
	data_byte_array:ARRAY[0..9] OF BYTE;
	i: INT;
END_VAR

fn_cyber_heartBeat := FALSE;

index := 0;
data_uint := STRING_TO_UINT(concat('16#',lac_str));
pDataOut[index] := ANY_TO_BYTE(data_uint/256);
index := index + 1;

pDataOut[index] := ANY_TO_BYTE(data_uint MOD 256);
index := index + 1;

data_uint := STRING_TO_UINT(concat('16#',cid_str));
pDataOut[index] := ANY_TO_BYTE(data_uint/256);
index := index + 1;

pDataOut[index] := ANY_TO_BYTE(data_uint MOD 256);
index := index + 1;

data_byte_array := Iccid_Get(ccid_str);
FOR i := 0 TO 9 DO
	pDataOut[index] := data_byte_array[i];
	index := index + 1;
END_FOR

pDataOut[index] := ANY_TO_BYTE(mins/256/256/256);
index := index + 1;

pDataOut[index] := ANY_TO_BYTE(mins/256/256);
index := index + 1;

pDataOut[index] := ANY_TO_BYTE(mins/256);
index := index + 1;

pDataOut[index] := ANY_TO_BYTE(mins);
index := index + 1;

pDataOut[index] := ANY_TO_BYTE(clientCode/256);
index := index + 1;

pDataOut[index] := ANY_TO_BYTE(clientCode);
index := index + 1;

pDataOut[index] := ANY_TO_BYTE(machineCode/256);
index := index + 1;

pDataOut[index] := ANY_TO_BYTE(machineCode);
index := index + 1;

pLenOut^ := index;

fn_cyber_heartBeat := TRUE;

END_FUNCTION

// MIC7001/Application/GPRS/Iccid_Get
FUNCTION Iccid_Get : ARRAY[0..9] OF BYTE
VAR_INPUT
	iccd :STRING;
END_VAR
VAR
	iccid_code :ARRAY[0..9] OF BYTE;
	
	byteHigh :BYTE := 0;
	byteLow :BYTE := 0;
	dstLen :INT := 0;
	
	srcIndex :INT := 0;
	bytesIndex :INT := 0;
	sub_str:STRING(32);
END_VAR

dstLen := len(iccd) / 2;

sub_str := iccd;
FOR bytesIndex := 0 TO dstLen - 1 DO
	iccid_code[bytesIndex] := BYTE_TO_BCD(STRING_TO_BYTE(left(sub_str,2)));	
	sub_str := delete(sub_str,2,1);
END_FOR

Iccid_Get := iccid_code;

END_FUNCTION

// MIC7001/Application/GPRS/fn_cyber_layer2
FUNCTION fn_cyber_layer2 : bool
VAR_INPUT
	dataType : BYTE := 0;
	paraId :BYTE := 0;
	dataIndex : UINT := 0;
	ver :BYTE := 1;
	res1 :BYTE := 0;
	LenIn :UINT := 0;
	pDataIn :POINTER TO BYTE;
	pLenOut :POINTER TO UINT;
	pDataOut :POINTER TO BYTE;
END_VAR
VAR
	i:UINT:= 0;
	index:UINT := 0;
END_VAR

fn_cyber_layer2 := FALSE;

index := 0;
pDataOut[index] := dataType;
index := index + 1;

pDataOut[index] := paraId;
index := index + 1;

pDataOut[index] := ANY_TO_BYTE(dataIndex/256);
index := index + 1;

pDataOut[index] := ANY_TO_BYTE(dataIndex MOD 256);
index := index + 1;

pDataOut[index] := ver;
index := index + 1;

pDataOut[index] := res1;
index := index + 1;

pDataOut[index] := ANY_TO_BYTE(LenIn/256);
index := index + 1;

pDataOut[index] := ANY_TO_BYTE(LenIn MOD 256);
index := index + 1;

FOR i := 0 TO LenIn-1 DO
	pDataOut[index] := pDataIn[i];
	index := index + 1;
END_FOR

pLenOut^ := index;

fn_cyber_layer2 := TRUE;
RETURN;

END_FUNCTION

// MIC7001/Application/GPRS/fn_sn_str_to_byte
FUNCTION fn_sn_str_to_byte : ARRAY[0..9] OF BYTE
VAR_INPUT
	sn:STRING(16);
END_VAR
VAR
	i: INT;
	bSN: ARRAY[0..9] OF BYTE;
	sub_str: STRING(255);
	num: UINT;
END_VAR

	
FOR i := 0 TO 2 DO
	bSN[i] := sn[i];
END_FOR

// 1.2 12
sub_str := mid(sn, 2, 4);
bSN[3] := STRING_TO_BYTE(sub_str);

// 1.3 34
sub_str := mid(sn, 2, 6);
bSN[4] := STRING_TO_BYTE(sub_str);

// 1.4 56
sub_str := mid(sn, 2, 8);
bSN[5] := STRING_TO_BYTE(sub_str);

// 1.5 78
sub_str := mid(sn, 2, 10);
bSN[6] := STRING_TO_BYTE(sub_str);

// 1.6 1234
sub_str := mid(sn, 4, 12);
num := STRING_TO_UINT(sub_str);
bSN[7] := ANY_TO_BYTE(num / 256);
bSN[8] := ANY_TO_BYTE(num MOD 256);

fn_sn_str_to_byte := bSN;

END_FUNCTION

// MIC7001/Application/GPRS/fn_cyber_layer1
FUNCTION fn_cyber_layer1 : bool
VAR_INPUT
	sn:POINTER TO BYTE;
	ver:BYTE := 0;
	lenIn:UINT := 0;
	pDataIn:POINTER TO BYTE;
	pLenOut:POINTER TO UINT ;
	pDataOut: POINTER TO BYTE;
END_VAR
VAR
	i:UINT;
	index:UINT;
	checksum:UINT;
END_VAR

fn_cyber_layer1 := FALSE;

index := 0;
checksum := 0;
FOR i := 0 TO 8 DO
	pDataOut[index] := sn[i];
	index := index+1;
	checksum := checksum + sn[i];
END_FOR

pDataOut[index] := ver;
index := index+1;
checksum := checksum + ver;

pDataOut[index] := ANY_TO_BYTE(lenIn/256);
index := index+1;
checksum := checksum + ANY_TO_BYTE(lenIn/256);

pDataOut[index] := ANY_TO_BYTE(lenIn MOD 256);
index := index+1;
checksum := checksum + ANY_TO_BYTE(lenIn MOD 256);

FOR i := 0 TO lenIn-1 DO
	pDataOut[index] := pDataIn[i];
	index := index+1;	
	checksum := checksum + pDataIn[i];
END_FOR

pDataOut[index] := ANY_TO_BYTE(checksum/256);
index := index+1;

pDataOut[index] := ANY_TO_BYTE(checksum MOD 256);
index := index+1;

pLenOut^ := index;

fn_cyber_layer1 := TRUE;

END_FUNCTION

// MIC7001/Application/GPRS/fb_m26
FUNCTION_BLOCK fb_m26
VAR_INPUT
	enable :BOOL := FALSE;
	ipaddr :STRING(32);
	port :UINT;
END_VAR
VAR_OUTPUT
	xBusy :BOOL := FALSE;
	xError :BOOL := FALSE;
	xDone :BOOL := FALSE;
	handle_m26 :CAA.HANDLE; 
END_VAR
VAR
	udp_init:Udp_Init;
	iStat :UINT := 0;
END_VAR

IF NOT enable THEN
	xBusy := FALSE;
	xError := FALSE;
	handle_m26 := 0;
	RETURN;
END_IF

CASE iStat OF
0:
	udp_init(xExecute := FALSE, ip_addr := ipaddr, port := port);
	udp_init.xExecute := TRUE;
	iStat := 10;
	
10:
	IF udp_init.xDone THEN
		xBusy := TRUE;
		handle_m26 := udp_init.udp_handle;
		iStat := 100;
	ELSIF udp_init.xError THEN
		iStat := 200;
	END_IF	

100:
	xDone:= TRUE;
	
200:
	xError := TRUE;

END_CASE


udp_init(ip_addr := ipaddr, port := port);

END_FUNCTION_BLOCK

// MIC7001/Application/gprs_lib/Udp_Init
FUNCTION_BLOCK Udp_Init
VAR_INPUT
	xExecute:BOOL := FALSE;
	ip_addr:STRING;
	port:UINT;
END_VAR
VAR_OUTPUT
	xDone :BOOL := FALSE;
	xError :BOOL := FALSE;
	xBusy :BOOL := FALSE;
	
	udp_handle :CAA.HANDLE; 
END_VAR
VAR
	udp_config_fb :Udp_Config;
	ComWrite: COM.Write;
	ComRead: COM.Read;	
	com_handle: CAA.HANDLE;
	init_start :DWORD := 0;
	iStat: INT := 0;
END_VAR

init_start := %ID48;
IF (init_start > 0) THEN
	RETURN;
END_IF

IF NOT xExecute THEN
	xDone := FALSE;
	xError := FALSE;
	xBusy := FALSE;
	iStat := 0;
	RETURN;
END_IF

CASE iStat OF
0:
	udp_config_fb(xExecute := FALSE,ip_addr := ip_addr, port := port, com_hand := com_handle); 
	iStat := 10;
	xBusy := TRUE;
10:
	udp_config_fb.xExecute := TRUE;
	IF udp_config_fb.xDone  THEN
		iStat := 100;
		xDone := TRUE;
		xBusy := FALSE;
		udp_handle := com_handle;
		ComWrite(xExecute := FALSE, hCom:= com_handle);
		ComRead(xExecute := FALSE, hCom:= com_handle);		
	ELSIF udp_config_fb.xError THEN
		xError := TRUE;
		iStat := 200;
	END_IF	
100: //succ

200: //error

END_CASE

udp_config_fb(ip_addr := ip_addr, port := port, com_hand := com_handle);

END_FUNCTION_BLOCK

// MIC7001/Application/gprs_lib/Udp_Config
FUNCTION_BLOCK Udp_Config
VAR_INPUT
	xExecute : BOOL := FALSE;
	ip_addr:STRING;
	port:UINT;
END_VAR
VAR_IN_OUT
	com_hand: CAA.HANDLE;
END_VAR
VAR_OUTPUT
	xDone : BOOL := FALSE;
	xError :BOOL := FALSE;
	xBusy : BOOL := FALSE;
END_VAR
VAR
	ton_fb :TON;
	Com1Params: 			ARRAY [1..7] OF COM.PARAMETER;	(* Settings to communicate with 
the COM Port *)
	ComOpen: 				COM.Open;
	ComClose: 				COM.Close;
	ComWrite: 				COM.Write;
	ComRead: 				COM.Read;	
	Rcv_Cnt: 				CAA.SIZE;
	xCom1CloseError: 		BOOL;
	xCom1WriteError: 		BOOL;
	xCom1ReadError: 		BOOL;
	uiComState: INT := 0;
	ComID:USINT:=6;

	position :INT := 0;
	at_cmd :STRING := 'AT$r';
	at_buffer :STRING;
	ate0_cmd :STRING := 'ATE0$r';
	ate0_buffer :STRING;
	cpin_cmd :STRING := 'AT+CPIN?$r';
	cpin_buffer :STRING;
	csq_cmd :STRING := 'AT+CSQ$r';
	csq_buffer :STRING;
	creg_cmd :STRING := 'AT+CREG?$r';
	creg_buffer :STRING;
	cgreg_cmd :STRING := 'AT+CGREG?$r';
	cgreg_buffer :STRING;
	qindi_cmd :STRING := 'AT+QINDI=1$r';
	qindi_buffer :STRING;     
	qimode_cmd :STRING := 'AT+QIMODE=0$r';
	qimode_buffer :STRING;     
	qifgcnt_cmd :STRING := 'AT+QIFGCNT=0$r';
	qifgcnt_buffer :STRING;
	qimux_cmd :STRING := 'AT+QIMUX=0$r';
	qimux_buffer :STRING;
	qicsgp_cmd :STRING := 'AT+QICSGP=1,$"CMNET$"$r';
	qicsgp_buffer :STRING;
	qideact_cmd :STRING := 'AT+QIDEACT$r';
	qideact_buffer :STRING;
	qiregapp_cmd :STRING := 'AT+QIREGAPP$r';
	qiregapp_buffer :STRING;
	qiact_cmd :STRING := 'AT+QIACT$r';
	qiact_buffer :STRING;
	qilocip_cmd :STRING := 'AT+QILOCIP$r';
	qilocip_buffer :STRING;
	qiopen_cmd :STRING := 'AT+QIOPEN=$"UDP$",$"';
	qiopen_buffer :STRING;
	loop_in_count :INT := 0;
	loop_out_count :INT := 0;
	
	reset_gprs_fb :reset_gprs;
END_VAR

IF NOT xExecute THEN
	xDone := FALSE;
	xError := FALSE;
	xBusy := FALSE;
	uiComState := 0;
	RETURN;
END_IF

CASE uiComState OF
	0:
	Com1Params[1].udiParameterId := COM.CAA_Parameter_Constants.udiPort;
	Com1Params[1].udiValue := ComID; 
	Com1Params[2].udiParameterId := COM.CAA_Parameter_Constants.udiBaudrate;
	Com1Params[2].udiValue := 115200;
	Com1Params[3].udiParameterId := COM.CAA_Parameter_Constants.udiParity;
	Com1Params[3].udiValue := INT_TO_UINT(COM.PARITY.NONE);
	Com1Params[4].udiParameterId := COM.CAA_Parameter_Constants.udiStopBits;
	Com1Params[4].udiValue := INT_TO_UINT(COM.STOPBIT.ONESTOPBIT);
	Com1Params[5].udiParameterId := COM.CAA_Parameter_Constants.udiTimeout;
	Com1Params[5].udiValue := 0;
	Com1Params[6].udiParameterId := COM.CAA_Parameter_Constants.udiByteSize;
	Com1Params[6].udiValue := 8;
	Com1Params[7].udiParameterId := COM.CAA_Parameter_Constants.udiBinary;
	Com1Params[7].udiValue := 0;					
	ComOpen(xExecute := TRUE, usiListLength:=UINT_TO_USINT(SIZEOF(Com1Params)/SIZEOF(COM.PARAMETER)),pParameterList:= ADR(Com1Params),hCom=> com_hand);			
	IF ComOpen.xError THEN
		uiComState := 32767;
	ELSIF ComOpen.xDone THEN
		uiComState := 1;
		com_hand := ComOpen.hCom;
		ComWrite(xExecute := FALSE,hCom:= com_hand);	
		ComRead(xExecute := FALSE,hCom:= com_hand);
	END_IF
	
	1:  // write "AT\r"
	ComWrite(xExecute := TRUE,hCom:= com_hand,pBuffer:= ADR(at_cmd),szSize:=len(at_cmd));		
	IF ComWrite.xError THEN
		uiComState := 32767;
	END_IF
	IF ComWrite.xDone THEN
		ComWrite(xExecute := FALSE, hCom:= com_hand);
		uiComState := 2;
	END_IF
	
	2:
	ton_fb(IN := TRUE, PT := TIME#300MS);
	IF (ton_fb.Q) THEN
		ton_fb(IN := FALSE, PT := TIME#300MS);
		uiComState := 3;
	END_IF
	
	3:
	ComRead(xExecute := TRUE,hCom:= com_hand, pBuffer:= ADR(at_buffer), szBuffer:= SIZEOF(at_buffer));			
	IF ComRead.xError THEN
		uiComState := 32767;
	END_IF
	IF ComRead.xDone THEN
		uiComState := 1;
		position := find(at_buffer, 'OK');
		IF position > 0 THEN
			uiComState := 4;
			loop_in_count := 0;
			loop_out_count := 0;
		END_IF
		ComRead(xExecute := FALSE, hCom:= com_hand);
	
		IF loop_out_count > 10 THEN
			uiComState := 32767;
			RETURN;
		END_IF
		
		// 通过gpio复位gprs模块
		loop_in_count := loop_in_count + 1;
		IF loop_in_count > 50 THEN
			loop_in_count := 0;
			loop_out_count := loop_out_count + 1;
			reset_gprs_fb(xExecute := FALSE);
			uiComState := 49;
			RETURN;
		END_IF
	END_IF
		
	4: // write "ATE0\r"
	ComWrite(xExecute := TRUE,hCom:= com_hand,pBuffer:= ADR(ate0_cmd),szSize:=len(ate0_cmd));		
	IF ComWrite.xError THEN
		uiComState := 32767;
	END_IF
	IF ComWrite.xDone THEN
		ComWrite(xExecute := FALSE, hCom:= com_hand);
		uiComState := 5;
	END_IF
	
	5:
	ton_fb(IN := TRUE, PT := TIME#300MS);
	IF (ton_fb.Q) THEN
		ton_fb(IN := FALSE, PT := TIME#300MS);
		uiComState := 6;
	END_IF
	
	6:
	ComRead(xExecute := TRUE,hCom:= com_hand, pBuffer:= ADR(ate0_buffer), szBuffer:= SIZEOF(ate0_buffer));			
	IF ComRead.xError THEN
		uiComState := 32767;
	END_IF
	IF ComRead.xDone THEN
		uiComState := 4;
		ComRead(xExecute := FALSE, hCom:= com_hand);
		position := find(ate0_buffer, 'OK');
		IF position > 0 THEN
			uiComState := 7;
		END_IF
	END_IF
	
	7: // write "AT+CPIN?\r"
	ComWrite(xExecute := TRUE,hCom:= com_hand,pBuffer:= ADR(cpin_cmd),szSize:=len(cpin_cmd));		
	IF ComWrite.xError THEN
		uiComState := 32767;
	END_IF
	IF ComWrite.xDone THEN
		ComWrite(xExecute := FALSE, hCom:= com_hand);
		uiComState := 8;
	END_IF
	
	8:
	ton_fb(IN := TRUE, PT := TIME#300MS);
	IF (ton_fb.Q) THEN
		ton_fb(IN := FALSE, PT := TIME#300MS);
		uiComState := 9;
	END_IF
	
	9:
	ComRead(xExecute := TRUE,hCom:= com_hand, pBuffer:= ADR(cpin_buffer), szBuffer:= SIZEOF(cpin_buffer));			
	IF ComRead.xError THEN
		uiComState := 32767;
	END_IF
	IF ComRead.xDone THEN
		uiComState := 7;
		ComRead(xExecute := FALSE, hCom:= com_hand);
		position := find(cpin_buffer, 'OK');
		IF position > 0 THEN
			uiComState := 10;
		END_IF
	END_IF
	
	10: // write "AT+CSQ\r"
	ComWrite(xExecute := TRUE,hCom:= com_hand,pBuffer:= ADR(csq_cmd),szSize:=len(csq_cmd));		
	IF ComWrite.xError THEN
		uiComState := 32767;
	END_IF
	IF ComWrite.xDone THEN
		ComWrite(xExecute := FALSE, hCom:= com_hand);
		uiComState := 11;
	END_IF
	
	11:
	ton_fb(IN := TRUE, PT := TIME#300MS);
	IF (ton_fb.Q) THEN
		ton_fb(IN := FALSE, PT := TIME#300MS);
		uiComState := 12;
	END_IF
	
	12:
	ComRead(xExecute := TRUE,hCom:= com_hand, pBuffer:= ADR(csq_buffer), szBuffer:= SIZEOF(csq_buffer));			
	IF ComRead.xError THEN
		uiComState := 32767;
	END_IF
	IF ComRead.xDone THEN
		uiComState := 10;
		ComRead(xExecute := FALSE, hCom:= com_hand);
		position := find(csq_buffer, 'OK');
		IF position > 0 THEN
			uiComState := 13;
		END_IF
	END_IF
	
	13: // write "AT+CREG?\r"
	ComWrite(xExecute := TRUE,hCom:= com_hand,pBuffer:= ADR(creg_cmd),szSize:=len(creg_cmd));		
	IF ComWrite.xError THEN
		uiComState := 32767;
	END_IF
	IF ComWrite.xDone THEN
		ComWrite(xExecute := FALSE, hCom:= com_hand);
		uiComState := 14;
	END_IF
	
	14:
	ton_fb(IN := TRUE, PT := TIME#300MS);
	IF (ton_fb.Q) THEN
		ton_fb(IN := FALSE, PT := TIME#300MS);
		uiComState := 15;
	END_IF
	
	15:
	ComRead(xExecute := TRUE,hCom:= com_hand, pBuffer:= ADR(creg_buffer), szBuffer:= SIZEOF(creg_buffer));			
	IF ComRead.xError THEN
		uiComState := 32767;
	END_IF
	IF ComRead.xDone THEN
		uiComState := 13;
		ComRead(xExecute := FALSE, hCom:= com_hand);
		position := find(creg_buffer, 'OK');
		IF position > 0 THEN
			uiComState := 16;
		END_IF
	END_IF
	
	16: // write "AT+CGREG?\r"
	ComWrite(xExecute := TRUE,hCom:= com_hand,pBuffer:= ADR(cgreg_cmd),szSize:=len(cgreg_cmd));		
	IF ComWrite.xError THEN
		uiComState := 32767;
	END_IF
	IF ComWrite.xDone THEN
		ComWrite(xExecute := FALSE, hCom:= com_hand);
		uiComState := 17;
	END_IF
	
	17:
	ton_fb(IN := TRUE, PT := TIME#300MS);
	IF (ton_fb.Q) THEN
		ton_fb(IN := FALSE, PT := TIME#300MS);
		uiComState := 18;
	END_IF
	
	18:
	ComRead(xExecute := TRUE,hCom:= com_hand, pBuffer:= ADR(cgreg_buffer), szBuffer:= SIZEOF(cgreg_buffer));			
	IF ComRead.xError THEN
		uiComState := 32767;
	END_IF
	IF ComRead.xDone THEN
		uiComState := 16;
		ComRead(xExecute := FALSE, hCom:= com_hand);
		position := find(cgreg_buffer, 'OK');
		IF position > 0 THEN
			uiComState := 19;
		END_IF
	END_IF
	
	19: // write "AT+QINDI=1\r"     
	ComWrite(xExecute := TRUE,hCom:= com_hand,pBuffer:= ADR(qindi_cmd),szSize:=len(qindi_cmd));		
	IF ComWrite.xError THEN
		uiComState := 32767;
	END_IF
	IF ComWrite.xDone THEN
		ComWrite(xExecute := FALSE, hCom:= com_hand);
		uiComState := 20;
	END_IF
	
	20:
	ton_fb(IN := TRUE, PT := TIME#300MS);
	IF (ton_fb.Q) THEN
		ton_fb(IN := FALSE, PT := TIME#300MS);
		uiComState := 21;
	END_IF
	
	21:
	ComRead(xExecute := TRUE,hCom:= com_hand, pBuffer:= ADR(qindi_buffer), szBuffer:= SIZEOF(qindi_buffer));			
	IF ComRead.xError THEN
		uiComState := 32767;
	END_IF
	IF ComRead.xDone THEN
		uiComState := 19;
		ComRead(xExecute := FALSE, hCom:= com_hand);
		position := find(qindi_buffer, 'OK');
		IF position > 0 THEN
			uiComState := 22;
			loop_in_count := 0;
			loop_out_count := 0;
		ELSE
			IF loop_out_count > 10 THEN
				uiComState := 32767;
				RETURN;
			END_IF
			
			// 通过gpio复位gprs模块
			loop_in_count := loop_in_count + 1;
			IF loop_in_count > 25 THEN
				loop_in_count := 0;
				loop_out_count := loop_out_count + 1;
				reset_gprs_fb(xExecute := FALSE);
				uiComState := 49;
				RETURN;
			END_IF
		END_IF
	END_IF
	
	22: // write "AT+QIMODE=0\r"     
	ComWrite(xExecute := TRUE,hCom:= com_hand,pBuffer:= ADR(qimode_cmd),szSize:=len(qimode_cmd));		
	IF ComWrite.xError THEN
		uiComState := 32767;
	END_IF
	IF ComWrite.xDone THEN
		ComWrite(xExecute := FALSE, hCom:= com_hand);
		uiComState := 23;
	END_IF
	
	23:
	ton_fb(IN := TRUE, PT := TIME#300MS);
	IF (ton_fb.Q) THEN
		ton_fb(IN := FALSE, PT := TIME#300MS);
		uiComState := 24;
	END_IF
	
	24:
	ComRead(xExecute := TRUE,hCom:= com_hand, pBuffer:= ADR(qimode_buffer), szBuffer:= SIZEOF(qimode_buffer));			
	IF ComRead.xError THEN
		uiComState := 32767;
	END_IF
	IF ComRead.xDone THEN
		uiComState := 22;
		ComRead(xExecute := FALSE, hCom:= com_hand);
		position := find(qimode_buffer, 'OK');
		IF position > 0 THEN
			uiComState := 25;
		ELSE
			IF loop_out_count > 10 THEN
				uiComState := 32767;
				RETURN;
			END_IF
			
			// 通过gpio复位gprs模块
			loop_in_count := loop_in_count + 1;
			IF loop_in_count > 25 THEN
				loop_in_count := 0;
				loop_out_count := loop_out_count + 1;
				reset_gprs_fb(xExecute := FALSE);
				uiComState := 49;
				RETURN;
			END_IF
		END_IF
		//uiComState := 25;
	END_IF
	
	25: // write "AT+QIFGCNT=0\r"     
	ComWrite(xExecute := TRUE,hCom:= com_hand,pBuffer:= ADR(qifgcnt_cmd),szSize:=len(qifgcnt_cmd));		
	IF ComWrite.xError THEN
		uiComState := 32767;
	END_IF
	IF ComWrite.xDone THEN
		ComWrite(xExecute := FALSE, hCom:= com_hand);
		uiComState := 26;
	END_IF
	
	26:
	ton_fb(IN := TRUE, PT := TIME#300MS);
	IF (ton_fb.Q) THEN
		ton_fb(IN := FALSE, PT := TIME#300MS);
		uiComState := 27;
	END_IF
	
	27:
	ComRead(xExecute := TRUE,hCom:= com_hand, pBuffer:= ADR(qifgcnt_buffer), szBuffer:= SIZEOF(qifgcnt_buffer));			
	IF ComRead.xError THEN
		uiComState := 32767;
	END_IF
	IF ComRead.xDone THEN
		uiComState := 25;
		ComRead(xExecute := FALSE, hCom:= com_hand);
		position := find(qifgcnt_buffer, 'OK');
		IF position > 0 THEN
			uiComState := 28;
		END_IF
	END_IF
	
	28: // write "AT+QIMUX=0\r"     
	ComWrite(xExecute := TRUE,hCom:= com_hand,pBuffer:= ADR(qimux_cmd),szSize:=len(qimux_cmd));		
	IF ComWrite.xError THEN
		uiComState := 32767;
	END_IF
	IF ComWrite.xDone THEN
		ComWrite(xExecute := FALSE, hCom:= com_hand);
		uiComState := 29;
	END_IF
	
	29:
	ton_fb(IN := TRUE, PT := TIME#300MS);
	IF (ton_fb.Q) THEN
		ton_fb(IN := FALSE, PT := TIME#300MS);
		uiComState := 30;
	END_IF
	
	30:
	ComRead(xExecute := TRUE,hCom:= com_hand, pBuffer:= ADR(qimux_buffer), szBuffer:= SIZEOF(qimux_buffer));			
	IF ComRead.xError THEN
		uiComState := 32767;
	END_IF
	IF ComRead.xDone THEN
		uiComState := 28;
		ComRead(xExecute := FALSE, hCom:= com_hand);
		position := find(qimux_buffer, 'OK');
		IF position > 0 THEN
			uiComState := 31;
		END_IF
		//uiComState := 31;
	END_IF
	
	31: // write "AT+QICSGP=1,\"CMNET\"\r"     
	ComWrite(xExecute := TRUE,hCom:= com_hand,pBuffer:= ADR(qicsgp_cmd),szSize:=len(qicsgp_cmd));		
	IF ComWrite.xError THEN
		uiComState := 32767;
	END_IF
	IF ComWrite.xDone THEN
		ComWrite(xExecute := FALSE, hCom:= com_hand);
		uiComState := 32;
	END_IF
	
	32:
	ton_fb(IN := TRUE, PT := TIME#300MS);
	IF (ton_fb.Q) THEN
		ton_fb(IN := FALSE, PT := TIME#300MS);
		uiComState := 33;
	END_IF
	
	33:
	ComRead(xExecute := TRUE,hCom:= com_hand, pBuffer:= ADR(qicsgp_buffer), szBuffer:= SIZEOF(qicsgp_buffer));			
	IF ComRead.xError THEN
		uiComState := 32767;
	END_IF
	IF ComRead.xDone THEN
		uiComState := 31;
		ComRead(xExecute := FALSE, hCom:= com_hand);
		position := find(qicsgp_buffer, 'OK');
		IF position > 0 THEN
			uiComState := 34;
		END_IF
	END_IF
	
	34: // write "AT+QIDEACT\r"     
	ComWrite(xExecute := TRUE,hCom:= com_hand,pBuffer:= ADR(qideact_cmd),szSize:=len(qideact_cmd));		
	IF ComWrite.xError THEN
		uiComState := 32767;
	END_IF
	IF ComWrite.xDone THEN
		ComWrite(xExecute := FALSE, hCom:= com_hand);
		uiComState := 35;
	END_IF
	
	35:
	ton_fb(IN := TRUE, PT := TIME#300MS);
	IF (ton_fb.Q) THEN
		ton_fb(IN := FALSE, PT := TIME#300MS);
		uiComState := 36;
	END_IF
	
	36:
	ComRead(xExecute := TRUE,hCom:= com_hand, pBuffer:= ADR(qicsgp_buffer), szBuffer:= SIZEOF(qicsgp_buffer));			
	IF ComRead.xError THEN
		uiComState := 32767;
	END_IF
	IF ComRead.xDone THEN
		uiComState := 34;
		ComRead(xExecute := FALSE, hCom:= com_hand);
		position := find(qicsgp_buffer, 'DEACT OK');
		IF position > 0 THEN
			uiComState := 37;
		END_IF
	END_IF
	
	37: // write "AT+QIREGAPP\r"     
	ComWrite(xExecute := TRUE,hCom:= com_hand,pBuffer:= ADR(qiregapp_cmd),szSize:=len(qiregapp_cmd));		
	IF ComWrite.xError THEN
		uiComState := 32767;
	END_IF
	IF ComWrite.xDone THEN
		ComWrite(xExecute := FALSE, hCom:= com_hand);
		uiComState := 38;
	END_IF
	
	38:
	ton_fb(IN := TRUE, PT := TIME#300MS);
	IF (ton_fb.Q) THEN
		ton_fb(IN := FALSE, PT := TIME#300MS);
		uiComState := 39;
	END_IF
	
	39:
	ComRead(xExecute := TRUE,hCom:= com_hand, pBuffer:= ADR(qiregapp_buffer), szBuffer:= SIZEOF(qiregapp_buffer));			
	IF ComRead.xError THEN
		uiComState := 32767;
	END_IF
	IF ComRead.xDone THEN
		uiComState := 37;
		ComRead(xExecute := FALSE, hCom:= com_hand);
		position := find(qiregapp_buffer, 'OK');
		IF position > 0 THEN
			uiComState := 40;
		END_IF
	END_IF
	
	40: // write "AT+QIACT\r"     
	ComWrite(xExecute := TRUE,hCom:= com_hand,pBuffer:= ADR(qiact_cmd),szSize:=len(qiact_cmd));		
	IF ComWrite.xError THEN
		uiComState := 32767;
	END_IF
	IF ComWrite.xDone THEN
		ComWrite(xExecute := FALSE, hCom:= com_hand);
		uiComState := 41;
	END_IF
	
	41:
	ton_fb(IN := TRUE, PT := TIME#300MS);
	IF (ton_fb.Q) THEN
		ton_fb(IN := FALSE, PT := TIME#300MS);
		uiComState := 42;
	END_IF
	
	42:
	ComRead(xExecute := TRUE,hCom:= com_hand, pBuffer:= ADR(qiact_buffer), szBuffer:= SIZEOF(qiact_buffer));			
	IF ComRead.xError THEN
		uiComState := 32767;
	END_IF
	IF ComRead.xDone THEN
		uiComState := 40;
		ComRead(xExecute := FALSE, hCom:= com_hand);
		position := find(qiact_buffer, 'OK');
		IF position > 0 THEN
			uiComState := 43;
		END_IF
	END_IF
	
	43: // write "AT+QILOCIP\r"     
	ComWrite(xExecute := TRUE,hCom:= com_hand,pBuffer:= ADR(qilocip_cmd),szSize:=len(qilocip_cmd));		
	IF ComWrite.xError THEN
		uiComState := 32767;
	END_IF
	IF ComWrite.xDone THEN
		ComWrite(xExecute := FALSE, hCom:= com_hand);
		uiComState := 44;
	END_IF
	
	44:
	ton_fb(IN := TRUE, PT := TIME#300MS);
	IF (ton_fb.Q) THEN
		ton_fb(IN := FALSE, PT := TIME#300MS);
		uiComState := 45;
	END_IF
	
	45:
	ComRead(xExecute := TRUE,hCom:= com_hand, pBuffer:= ADR(qilocip_buffer), szBuffer:= SIZEOF(qilocip_buffer));			
	IF ComRead.xError THEN
		uiComState := 32767;
	END_IF
	IF ComRead.xDone THEN
		uiComState := 46;
		ComRead(xExecute := FALSE, hCom:= com_hand);
		position := find(qilocip_buffer, 'ERROR');
		IF position > 0 THEN
			uiComState := 43;
		END_IF
	END_IF
	
	46: // write "AT+QIOPEN=\"UDP\",\"47.107.240.29\",123456\r"  
	qiopen_cmd := concat(qiopen_cmd, ip_addr);
	qiopen_cmd := concat(qiopen_cmd, '$",');
	qiopen_cmd := concat(qiopen_cmd, ANY_TO_STRING(port));
	qiopen_cmd := concat(qiopen_cmd, '$r');   
	ComWrite(xExecute := TRUE,hCom:= com_hand,pBuffer:= ADR(qiopen_cmd),szSize:=len(qiopen_cmd));		
	IF ComWrite.xError THEN
		uiComState := 32767;
	END_IF
	IF ComWrite.xDone THEN
		ComWrite(xExecute := FALSE, hCom:= com_hand);
		uiComState := 47;
	END_IF
	
	47:
	ton_fb(IN := TRUE, PT := TIME#300MS);
	IF (ton_fb.Q) THEN
		ton_fb(IN := FALSE, PT := TIME#300MS);
		uiComState := 48;
	END_IF
	
	48:
	ComRead(xExecute := TRUE,hCom:= com_hand, pBuffer:= ADR(qiopen_buffer), szBuffer:= SIZEOF(qiopen_buffer));			
	IF ComRead.xError THEN
		uiComState := 32767;
	END_IF
	IF ComRead.xDone THEN
		uiComState := 46;
		ComRead(xExecute := FALSE, hCom:= com_hand);
		position := find(qiopen_buffer, 'CONNECT OK');
		IF position > 0 THEN
			uiComState := 255;
		ELSE
			position := find(qiopen_buffer, 'ALREAY CONNECT');
			IF position > 0 THEN
				uiComState := 255;
			END_IF
		END_IF
	END_IF
	
	49:
	reset_gprs_fb.xExecute := TRUE;
	IF reset_gprs_fb.xDone THEN
		uiComState := 1;
	END_IF
	
	255:
		xDone := TRUE;
		
	32767:	
		xError := TRUE;
END_CASE

reset_gprs_fb();

END_FUNCTION_BLOCK

// MIC7001/Application/gprs_lib/reset_gprs
FUNCTION_BLOCK reset_gprs
VAR_INPUT
	xExecute:BOOL := FALSE;
END_VAR
VAR_OUTPUT
	xDone : BOOL := FALSE;
	xError :BOOL := FALSE;
	xBusy :BOOL := FALSE;
END_VAR
VAR
	iState :INT := 0;
	ton_fb :TON; 
END_VAR

IF NOT xExecute THEN
	iState := 0;
	xDone := FALSE;
	xBusy := FALSE;
	xError := FALSE;
	RETURN;
END_IF

CASE iState OF
0:
	xBusy := TRUE;
	set_gpio_value(129, 1);
	iState := 10;
	
10:
	ton_fb(IN := TRUE, PT := TIME#2000MS);
	IF (ton_fb.Q) THEN
		ton_fb(IN := FALSE, PT := TIME#2000MS);
		iState := 20;
	END_IF
	
20:
	set_gpio_value(129, 0);
	iState := 30;
	
30:
	ton_fb(IN := TRUE, PT := TIME#5000MS);
	IF (ton_fb.Q) THEN
		ton_fb(IN := FALSE, PT := TIME#5000MS);
		iState := 40;
	END_IF
	
40:
	iState := 255;	
	
255:
	xDone := TRUE;
	xBusy := FALSE;
32767:
	xError := TRUE;
END_CASE

END_FUNCTION_BLOCK

// MIC7001/Application/gprs_lib/Udp_Write
FUNCTION_BLOCK Udp_Write
VAR_INPUT
	xExecute :BOOL := FALSE;
	com :CAA.HANDLE;
	buffer: CAA.PVOID;
	size :CAA.SIZE;
END_VAR
VAR_OUTPUT
	xDone :BOOL := FALSE;
	xBusy :BOOL := FALSE;
	xError :BOOL := FALSE;
	atcState :INT;
END_VAR
VAR
	ComWrite: COM.Write;
	ComRead: COM.Read;	
	qisend_buffer :STRING := 'AT+QISEND='; 
	ton_fb :TON;  
	ack_buffer1 :STRING;
	ack_buffer2 :STRING;
	position :INT := -1;
	end_flag :ARRAY[0..1] OF BYTE;
	actionState :INT := 0;
	loop_count1 :INT := 0;
	loop_count2 :INT := 0;
	read_data_buffer: ARRAY[0..1499] OF BYTE;
END_VAR

IF NOT xExecute OR com = 0 THEN
	xDone := FALSE;
	xError := FALSE;
	xBusy := FALSE;
	actionState := 0;
	qisend_buffer := 'AT+QISEND='; 
	ComWrite(xExecute := FALSE);
	ComRead(xExecute := FALSE);
	RETURN;
END_IF

CASE actionState OF
0:
	ComRead(xExecute := TRUE,hCom:= com, pBuffer:= ADR(read_data_buffer), szBuffer:= SIZEOF(read_data_buffer));			
	IF ComRead.xError THEN
		ComRead(xExecute := FALSE);		
		actionState := 32767;
	END_IF
	IF ComRead.xDone THEN
		ComRead(xExecute := FALSE);			
		actionState := 1;
	END_IF

1:
	qisend_buffer := concat(qisend_buffer, ANY_TO_STRING(size));
	qisend_buffer := concat(qisend_buffer, '$r'); 
	actionState := 5;
	
5:
	ComWrite(xExecute := TRUE, hCom:= com, pBuffer:= ADR(qisend_buffer), szSize:= len(qisend_buffer));
	IF ComWrite.xError THEN
		actionState := 32767;
	END_IF
	IF ComWrite.xDone THEN
		actionState := 10;
		ComWrite(xExecute := FALSE, hCom:= com);	
	END_IF
	
10:
	ton_fb(IN := TRUE, PT := TIME#200MS);
	IF (ton_fb.Q) THEN
		ton_fb(IN := FALSE, PT := TIME#200MS);
		actionState := 20;
		ComRead(xExecute := FALSE);		
	END_IF
	
20:
	ComRead(xExecute := TRUE,hCom:= com, pBuffer:= ADR(ack_buffer1), szBuffer:= SIZEOF(ack_buffer1));			
	IF ComRead.xError THEN
		atcState := 32767;
	END_IF
	IF ComRead.xDone THEN
		
		position := find(ack_buffer1, '>');
		IF position > 0 THEN
			actionState := 30;
		ELSE
			actionState := 10;
		END_IF
		ComRead(xExecute := FALSE, hCom:= com);
		
		loop_count1 := loop_count1 + 1;
		IF loop_count1 > 50 THEN
			loop_count1 := 0;
			actionState := 32767;
		END_IF
	END_IF
	
30:
	ComWrite(xExecute := TRUE, hCom:= com, pBuffer:= buffer, szSize:= size);
	IF ComWrite.xError THEN
		actionState := 32767;
	END_IF
	IF ComWrite.xDone THEN
		actionState := 40;
		ComWrite(xExecute := FALSE, hCom:= com);	
	END_IF
	
40:
	end_flag[0] := 16#1A;
	ComWrite(xExecute := TRUE, hCom:= com, pBuffer:= ADR(end_flag), szSize:= 1);
	IF ComWrite.xError THEN
		actionState := 32767;
	END_IF
	IF ComWrite.xDone THEN
		actionState := 50;
		ComWrite(xExecute := FALSE, hCom:= com);	
	END_IF
	
50:
	ton_fb(IN := TRUE, PT := TIME#300MS);
	IF (ton_fb.Q) THEN
		ton_fb(IN := FALSE, PT := TIME#300MS);
		actionState := 60;
	END_IF
	
60:
	ComRead(xExecute := TRUE,hCom:= com, pBuffer:= ADR(ack_buffer2), szBuffer:= SIZEOF(ack_buffer2));			
	IF ComRead.xError THEN
		atcState := 32767;
	END_IF
	IF ComRead.xDone THEN
		position := find(ack_buffer2, 'SEND OK');
		IF position > 0 THEN
			actionState := 255;
		ELSE
			actionState := 50;
		END_IF
		ComRead(xExecute := FALSE, hCom:= com);
		loop_count2 := loop_count2 + 1;
		IF loop_count2 > 50 THEN
			loop_count2 := 0;
			actionState := 32767;
		END_IF
	END_IF
	
255:
	xDone := TRUE;
	xError := FALSE;
	xBusy := FALSE;
	actionState := 250;

	loop_count1 := 0;
	loop_count2 := 0; 
	ack_buffer1 := '';
	ack_buffer2 := '';
	qisend_buffer := 'AT+QISEND=';	
	
250:

32767:
	xDone := FALSE;
	xError := TRUE;
	xBusy := FALSE;
	actionState := 32700;

	loop_count1 := 0;
	loop_count2 := 0; 
	ack_buffer1 := '';
	ack_buffer2 := '';
	qisend_buffer := 'AT+QISEND=';	
	
32700:

END_CASE

END_FUNCTION_BLOCK

// MIC7001/Application/gprs_lib/UDP_Read
FUNCTION_BLOCK UDP_Read
VAR_INPUT
	xExecute:BOOL := FALSE;
	com :CAA.HANDLE;
	buffer: CAA.PVOID;
	rsize : CAA.SIZE;
END_VAR
VAR_OUTPUT
	xDone :BOOL := FALSE;
	xBusy :BOOL := FALSE;
	xError :BOOL := FALSE;
	size :CAA.SIZE;
	
END_VAR
VAR
	ton_fb :TON;  
	ComWrite: COM.Write;
	ComRead: COM.Read;	
	ack_buffer :STRING[1499];
	//ack_buffer :ARRAY[0..1499] OF BYTE;
	position :INT := -1;
	qird :STRING := 'AT+QIRD=0,1,0,1500$R';

	read_data_buffer: ARRAY[0..1499] OF BYTE;
	read_tmp_buffer: ARRAY[0..1499] OF BYTE;
	i :INT;
	read_num :INT;
	comma1 :INT;
	comma2 :INT;
	new_line :INT;
	data_len :INT := 0;
	//uchar *pos, *comma1, *comma2, *new_line;
	
	loop_count :INT := 0;
	loop_exit :INT := 0;
	
	del_atcState :INT;
	iStat :UINT := 0;
END_VAR

IF com = 0 OR NOT xExecute THEN
	xDone := FALSE;
	xError := FALSE;
	xBusy := FALSE;
	iStat := 0;
	position := -1;
	size := 0;
	ComRead(xExecute := FALSE);
	RETURN;
END_IF

CASE iStat OF
	0:
	ComRead(xExecute := TRUE,hCom:= com, pBuffer:= ADR(ack_buffer), szBuffer:= SIZEOF(ack_buffer));			
	IF ComRead.xError THEN
		ComRead(xExecute := FALSE, hCom:= com);
		iStat := 32767;
	END_IF
	
	IF ComRead.xDone THEN
		position := find(ack_buffer, '+QIRDI: 0,1,0');
		IF position > 0 THEN
			iStat := 2;
		ELSE
			iStat := 1;
		END_IF
		ComRead(xExecute := FALSE, hCom:= com);
		loop_count := loop_count + 1;
		IF loop_count > 20 THEN
			iStat := 2;
			loop_count := 0;
		END_IF
	END_IF
	
	1:
	ton_fb(IN := TRUE, PT := TIME#300MS);
	IF (ton_fb.Q) THEN
		ton_fb(IN := FALSE, PT := TIME#300MS);
		iStat := 0;
	END_IF
	
	2:
	ComWrite(xExecute := TRUE, hCom:= com, pBuffer:= ADR(qird), szSize:= len(qird));
	IF ComWrite.xError THEN
		iStat := 32767;
	END_IF
	
	IF ComWrite.xDone THEN
		iStat := 3;
		ComWrite(xExecute := FALSE, hCom:= com);	
	END_IF
	
	3:
	ton_fb(IN := TRUE, PT := TIME#300MS);
	IF (ton_fb.Q) THEN
		ton_fb(IN := FALSE, PT := TIME#300MS);
		iStat := 4;
	END_IF
	
	4:
	ComRead(xExecute := TRUE,hCom:= com, pBuffer:= ADR(read_data_buffer), szBuffer:= rsize);			
	IF ComRead.xError THEN
		iStat := 32767;
	END_IF
	IF ComRead.xDone THEN
		iStat := 5;
		read_num :=  ANY_TO_INT(ComRead.szSize);
		ComRead(xExecute := FALSE, hCom:= com);		
	END_IF
	
	5: //查找第一个逗号，第二次读取的时候，会返回OK，表示已经读完
	IF read_num = 6 THEN
		iStat := 0;
		loop_exit := loop_exit + 1;
		IF loop_exit > 1 THEN
			loop_exit := 0;
			iStat := 32767;
		END_IF
		RETURN;
	END_IF
	FOR i := 0 TO read_num - 1 BY 1 DO
		iStat := 32767;
		IF read_data_buffer[i] = 16#2C THEN
			comma1 := i;
			iStat := 6;
			RETURN;
		END_IF
	END_FOR;
	
	6: //查找第二个逗号
	FOR i := comma1 + 1 TO read_num - 1 BY 1 DO
		iStat := 32767;
		IF read_data_buffer[i] = 16#2C THEN
			comma2 := i;
			iStat := 7;
			RETURN;
		END_IF
	END_FOR;
	
	7: //查找回车换行
	FOR i := comma2 + 1 TO read_num - 1 BY 1 DO
		iStat := 32767;
		IF read_data_buffer[i] = 16#0D  AND read_data_buffer[i + 1] = 16#0A THEN
			new_line := i;
			iStat := 8;
			RETURN;
		END_IF
	END_FOR;
	
	8: // 获取数据长度
	FOR i := comma2 + 1 TO new_line - 1 BY 1 DO
		data_len := data_len *10 + read_data_buffer[i] - 16#30;
	END_FOR;

	iStat := 255;
	IF data_len > 0 THEN
		size := data_len;
		SysMemCpy(pDest:=buffer,pSrc:=ADR(read_data_buffer) + new_line + 2, udiCount:=data_len);
		
		data_len := 0;
		ack_buffer := '';
		loop_count := 0;
		read_num := 0;
		FOR i := 0 TO 1499 BY 1 DO
			read_data_buffer[i] := 0;
		END_FOR
	END_IF
	
	255:
		ComRead(xExecute := FALSE);
		xDone := TRUE;
		xBusy := FALSE;
		xError := FALSE;
		iStat := 256;
		
		data_len := 0;
		ack_buffer := '';
		loop_count := 0;
		read_num := 0;
		FOR i := 0 TO 1499 BY 1 DO
			read_data_buffer[i] := 0;
		END_FOR		
	256:
	
	32767:
		ComRead(xExecute := FALSE);
		xError := TRUE;
		xDone := FALSE;
		xBusy := FALSE;
		iStat := 32700;
		
		data_len := 0;
		ack_buffer := '';
		loop_count := 0;
		read_num := 0;
		FOR i := 0 TO 1499 BY 1 DO
			read_data_buffer[i] := 0;
		END_FOR		
	32700:
	
END_CASE

END_FUNCTION_BLOCK

// MIC7001/Application/GPRS/File_Read
FUNCTION_BLOCK File_Read
VAR_INPUT
	file_name :STRING;
END_VAR
VAR_OUTPUT
	sReadLine		: STRING;
	isRead          :BOOL := FALSE;	
END_VAR
VAR
	hfile			: CAA.HANDLE;
	FileOpen 		: File.Open;
	FileClose		: File.Close;
	FileRead		: File.Read;
	
	iState			: UINT := 0;	
	xError			: BOOL := FALSE;
END_VAR

 CASE iState OF
	0: // Open the file again, with read access.
	   isRead := false;
	   FileOpen(xExecute:= TRUE, sFileName:= file_name, xExclusive:= FALSE, eFileMode:= File.MODE.MREAD);
	   IF FileOpen.xDone = TRUE THEN
		   hfile := FileOpen.hFile;
		   FileOpen(xExecute:= FALSE);
		   iState := 1;
		   sReadLine := '';
	   ELSIF FileOpen.xError = TRUE THEN
		   iState:= 32767;
		   FileOpen(xExecute:= FALSE);
	   END_IF

	1: // Read the string from the file.
	   FileRead(xExecute:= TRUE, hFile:= hfile, pBuffer:= ADR(sReadLine), szBuffer:= SIZEOF(sReadLine));
	   IF FileRead.xDone = TRUE THEN
		   iState := 2;		   
		   sReadLine := MID(sReadLine, ANY_TO_INT(FileRead.szSize), 1);
		   FileRead(xExecute:= FALSE);
	   ELSIF FileRead.xError = TRUE THEN
		   iState:= 32767;
		   FileRead(xExecute:= FALSE);
	   END_IF 
	   
	 2: // Close that file.
	   FileClose(xExecute:= TRUE, hFile:= hfile);
	   IF FileClose.xDone = TRUE THEN
		   iState := 3;
		   FileClose(xExecute:= FALSE);
	   ELSIF FileClose.xError = TRUE THEN
		   iState:= 32767;
		   FileClose(xExecute:= FALSE);
	   END_IF
	   
	3: 	  
		isRead := TRUE;
		iState := 0;
		
	32767: 		
	
END_CASE

END_FUNCTION_BLOCK

// MIC7001/Application/gprs_lib/Com_Read
FUNCTION_BLOCK Com_Read
VAR_INPUT
	xExecute:BOOL := FALSE;
	com :CAA.HANDLE;
	wbuffer: CAA.PVOID;
	wsize :CAA.SIZE;	
	rbuffer: CAA.PVOID;
	rsize : CAA.SIZE;
END_VAR
VAR_OUTPUT
	xDone:BOOL := FALSE;
	xBusy:BOOL := FALSE;
	xError:BOOL := FALSE;
	size :CAA.SIZE;
END_VAR
VAR
	iState :INT;
	ton_fb :TON;  
	ComWrite: COM.Write;
	ComRead: COM.Read;	
	actionState :INT;
END_VAR

IF NOT xExecute THEN
	iState := 0;
	xDone := FALSE;
	xBusy := FALSE;
	xError := FALSE;
	size := 0;
	RETURN;
END_IF

CASE iState OF
0:
	size := 0;
	ComWrite(xExecute := TRUE, hCom:= com, pBuffer:= wbuffer, szSize:= wsize);
	IF ComWrite.xError THEN
		iState := 32767;
	END_IF
	IF ComWrite.xDone THEN
		iState := 10;
		ComWrite(xExecute := FALSE, hCom:= com);	
	END_IF
	xBusy := TRUE;
	
10:
	ton_fb(IN := TRUE, PT := TIME#300MS);
	IF (ton_fb.Q) THEN
		ton_fb(IN := FALSE, PT := TIME#300MS);
		iState := 20;
	END_IF
	
20:
	ComRead(xExecute := TRUE,hCom:= com, pBuffer:= rbuffer, szBuffer:= rsize);			
	IF ComRead.xError THEN
		iState := 32767;
	END_IF
	IF ComRead.xDone THEN
		iState := 255;
		size := ComRead.szSize;
		ComRead(xExecute := FALSE, hCom:= com);		
	END_IF
	
255:
	xDone := TRUE;
	xBusy := FALSE;
	
32767:
	xError := TRUE;
	
END_CASE

END_FUNCTION_BLOCK

// MIC7001/Application/GPRS/fb_get_iccid
FUNCTION_BLOCK fb_get_iccid
VAR_INPUT
	xExecute:BOOL := FALSE;
	m26_handle:CAA.HANDLE; 
END_VAR

VAR_OUTPUT
	iccid:STRING(32);
	xDone:BOOL := FALSE;
	xBusy :BOOL := FALSE;
	xError:BOOL := FALSE;
END_VAR

VAR
	iStat:UINT := 0;
	udp_handle :CAA.HANDLE; 
	accid_cmd :STRING := 'AT+ICCID$r';
	iccid_read_buffer :STRING(255);
	com_read :Com_Read;
	udp_init_fb: INT;
	size:CAA.SIZE;
	position :INT := -1;
	ICCID_HEAD:STRING := '+ICCID: ';
	timer01:ton;
END_VAR


IF NOT xExecute OR m26_handle = 0 THEN
	xDone := FALSE;
	xBusy := FALSE;
	xError := FALSE;
	iccid := '';
	iStat := 0;
	RETURN;
END_IF 		

IF iccid <> '' THEN  //已经读到了，不需再读
	xDone := TRUE;
	xBusy := FALSE;
	xError := FALSE;
	RETURN; 
END_IF

CASE iStat OF
0:
	com_read(xExecute := FALSE);
	iStat := 10;
	timer01(in := FALSE);
	com_read.xExecute := TRUE;
10:
	IF com_read.xDone THEN
		IF com_read.size > 0 THEN
			position := find(iccid_read_buffer, ICCID_HEAD);
			IF position > 0 THEN
				iccid := mid(iccid_read_buffer, 20, position + len(ICCID_HEAD));
				xDone := TRUE;
				iStat := 100;
			END_IF
		END_IF
	ELSIF com_read.xError THEN
		xDone := FALSE;
		iStat := 200;
	END_IF	
	timer01(in := NOT timer01.Q, pt := T#2S);
	IF timer01.Q THEN
		iStat := 0;
	END_IF
100:

200:

END_CASE

com_read(com:= m26_handle, wbuffer:= ADR(accid_cmd), wsize := len(accid_cmd), rbuffer := ADR(iccid_read_buffer), rsize := SIZEOF(iccid_read_buffer));

END_FUNCTION_BLOCK

// MIC7001/Application/GPRS/fb_get_lac
FUNCTION_BLOCK fb_get_lac
VAR_INPUT
	xExecute:BOOL := FALSE;
	m26_handle:CAA.HANDLE; 
END_VAR
VAR_OUTPUT
	lac:STRING(4) := '0000';
	ci :STRING(4) := '0000';
	xDone:BOOL := FALSE;
	xError:BOOL := FALSE;
END_VAR
VAR
	iStat:UINT := 0;
	udp_handle :CAA.HANDLE; 
	lac_set_cmd :STRING := 'AT+CREG=2$r';
	lac_get_cmd :STRING := 'AT+CREG?$r';
	lac_close_cmd :STRING := 'AT+CREG=0$r';
	lac_read_buffer :STRING(255);
	com_read :Com_Read;
	udp_init_fb: INT;
	size:CAA.SIZE;
	position :INT := -1;
	LACID_HEAD:STRING := '+CREG:';
	lac_str:STRING(8);
	ci_str:STRING(8);
	cntr: INT;
END_VAR


IF m26_handle = 0 THEN
	RETURN;
END_IF

IF NOT xExecute THEN
	xDone := FALSE;
	xError := FALSE;
	lac := '0000';
	ci := '0000';
	iStat := 0;
	
	RETURN;
END_IF 		

CASE iStat OF
0:
	com_read(xExecute := FALSE);
	com_read.wbuffer:= ADR(lac_set_cmd);
 	com_read.wsize := len(lac_set_cmd);
	com_read.xExecute := TRUE;	
	iStat := 5;
5:  //set m26 for lac and ci with command:  AT+CREG=2
	IF com_read.xDone THEN
		size := com_read.size;
		IF size > 0 THEN
			position := find(lac_read_buffer, 'OK');
			IF position > 0 THEN
				com_read(xExecute := FALSE);
				com_read.wbuffer:= ADR(lac_get_cmd);
				com_read.wsize := len(lac_get_cmd);
				com_read.xExecute := TRUE;				
				iStat := 10;
				cntr := 0;
			END_IF
		ELSE
			iStat := 0;
		END_IF
	ELSIF com_read.xError THEN
		xDone := FALSE;
	END_IF	

10:  //read lac and ci with command: AT+CREG?
	IF com_read.xDone THEN
		IF com_read.size > 0 THEN
			position := find(lac_read_buffer, LACID_HEAD);
			IF position > 0 THEN
				position := find(lac_read_buffer, '$"');
				IF position > 0 THEN
					lac := mid(lac_read_buffer, 4, position + 1);
					ci := mid(lac_read_buffer, 4, position + 8);
					iStat := 20;
					size := 0;
					com_read(xExecute := FALSE);
					com_read.wbuffer:= ADR(lac_close_cmd);
 					com_read.wsize := len(lac_close_cmd);
					com_read.xExecute := TRUE;
				END_IF
			ELSE
				iStat := 0;
			END_IF
		END_IF
		cntr := cntr + 1;
		IF cntr > 50 THEN
			iStat := 0;
		END_IF
	ELSIF com_read.xError THEN
		xDone := FALSE;
	END_IF	
	
20:  //close
	IF com_read.xDone THEN
		size := com_read.size;
		IF size > 0 THEN
			position := find(lac_read_buffer, 'OK');
			IF position > 0 THEN
				iStat := 100;
				xDone := TRUE;
			END_IF
		ELSE
			xDone := FALSE;
		END_IF
	ELSIF com_read.xError THEN
		xDone := FALSE;
	END_IF	
100: //ok

END_CASE

